// ---- DUTs/IO/Topology/RC40_A3_EK1122_E505EE87.TcDUT
{attribute 'GeneratedUsingTerminal: EK1122-0000-0018'}
{attribute addProperty BoxType "EK1122-0000-0018"}
{attribute addProperty Id "RC40_EPP_EPP1322_0001RC40_EPP_EPP1322_0001_ECA1E6F9120"}
{attribute addProperty CRC "3842371207"}
{attribute addProperty Size "120"}
{attribute addProperty Name "RC40_A3 (EK1122)"}
TYPE RC40_A3_EK1122_E505EE87 EXTENDS EK1122_1FC0878B :
STRUCT
    {attribute addProperty Name "RC40_EPP (EPP1322-0001)"}
    {attribute addProperty PreviousPort "RC40_A3 (EK1122) : D"}
    {attribute addProperty SyncUnit "default"}
    RC40_EPP_EPP1322_0001 : RC40_EPP_EPP1322_0001_ECA1E6F9;
END_STRUCT
END_TYPE

// ---- DUTs/IO/Topology/RC40_1_EK1100_B918F64D.TcDUT
{attribute 'GeneratedUsingTerminal: EK1100-0000-0018'}
{attribute addProperty BoxType "EK1100-0000-0018"}
{attribute addProperty Id "RC40_A2_EK1122RC40_A2_EK1122_EAFADCC873RC40_A3_EK1122RC40_A3_EK1122_E505EE87120RC40_A5_EL1809EL1809_32157CFD20RC40_A6_EL1809EL1809_32157CFD20RC40_A7_EL2809EL2809_2B6483BD19RC40_A8_EL2809EL2809_2B6483BD19RC40_A9_EL2809EL2809_2B6483BD19RC40_1_EndTerminal_EL9010EL9010_D29C20850"}
{attribute addProperty CRC "3105420877"}
{attribute addProperty Size "290"}
{attribute addProperty Name "RC40_1 (EK1100)"}
TYPE RC40_1_EK1100_B918F64D EXTENDS EK1100_1FC0878B :
STRUCT
    {attribute addProperty Name "RC40_A2 (EK1122)"}
    {attribute addProperty PreviousPort "RC40_1 (EK1100) : B"}
    {attribute addProperty SyncUnit "default"}
    RC40_A2_EK1122 : RC40_A2_EK1122_EAFADCC8;
    {attribute addProperty Name "RC40_A3 (EK1122)"}
    {attribute addProperty PreviousPort "RC40_A2 (EK1122) : C"}
    {attribute addProperty SyncUnit "default"}
    RC40_A3_EK1122 : RC40_A3_EK1122_E505EE87;
    {attribute addProperty Name "RC40_A5 (EL1809)"}
    {attribute addProperty PreviousPort "RC40_A3 (EK1122) : C"}
    {attribute addProperty SyncUnit "C40"}
    RC40_A5_EL1809 : EL1809_32157CFD;
    {attribute addProperty Name "RC40_A6 (EL1809)"}
    {attribute addProperty PreviousPort "RC40_A5 (EL1809) : B"}
    {attribute addProperty SyncUnit "C40"}
    RC40_A6_EL1809 : EL1809_32157CFD;
    {attribute addProperty Name "RC40_A7 (EL2809)"}
    {attribute addProperty PreviousPort "RC40_A6 (EL1809) : B"}
    {attribute addProperty SyncUnit "C40"}
    RC40_A7_EL2809 : EL2809_2B6483BD;
    {attribute addProperty Name "RC40_A8 (EL2809)"}
    {attribute addProperty PreviousPort "RC40_A7 (EL2809) : B"}
    {attribute addProperty SyncUnit "C40"}
    RC40_A8_EL2809 : EL2809_2B6483BD;
    {attribute addProperty Name "RC40_A9 (EL2809)"}
    {attribute addProperty PreviousPort "RC40_A8 (EL2809) : B"}
    {attribute addProperty SyncUnit "C40"}
    RC40_A9_EL2809 : EL2809_2B6483BD;
    {attribute addProperty Name "RC40_1_EndTerminal (EL9010)"}
    {attribute addProperty PreviousPort "RC40_A9 (EL2809) : B"}
    {attribute addProperty SyncUnit "default"}
    RC40_1_EndTerminal_EL9010 : EL9010_D29C2085;
END_STRUCT
END_TYPE

// ---- DUTs/IO/Topology/RC40_2_EK1100_ACF07759.TcDUT
{attribute 'GeneratedUsingTerminal: EK1100-0000-0018'}
{attribute addProperty BoxType "EK1100-0000-0018"}
{attribute addProperty Id "RC40_B1_EL7041_1000EL7041_86DE63E743RC40_B2_EL7041_1000EL7041_86DE63E743RC40_C11_EL7041_1000EL7041_86DE63E743RC40_C12_EL7041_1000EL7041_86DE63E743RC40_C21_EL7041_1000EL7041_86DE63E743RC40_C22_EL7041_1000EL7041_86DE63E743RC40_2_EndTerminal_EL9010EL9010_D29C20850"}
{attribute addProperty CRC "2901440345"}
{attribute addProperty Size "258"}
{attribute addProperty Name "RC40_2 (EK1100)"}
TYPE RC40_2_EK1100_ACF07759 EXTENDS EK1100_1FC0878B :
STRUCT
    {attribute addProperty Name "RC40_B1 (EL7041-1000)"}
    {attribute addProperty PreviousPort "RC40_2 (EK1100) : B"}
    {attribute addProperty SyncUnit "C40"}
    RC40_B1_EL7041_1000 : EL7041_86DE63E7;
    {attribute addProperty Name "RC40_B2 (EL7041-1000)"}
    {attribute addProperty PreviousPort "RC40_B1 (EL7041-1000) : B"}
    {attribute addProperty SyncUnit "C40"}
    RC40_B2_EL7041_1000 : EL7041_86DE63E7;
    {attribute addProperty Name "RC40_C11 (EL7041-1000)"}
    {attribute addProperty PreviousPort "RC40_B2 (EL7041-1000) : B"}
    {attribute addProperty SyncUnit "C40"}
    RC40_C11_EL7041_1000 : EL7041_86DE63E7;
    {attribute addProperty Name "RC40_C12 (EL7041-1000)"}
    {attribute addProperty PreviousPort "RC40_C11 (EL7041-1000) : B"}
    {attribute addProperty SyncUnit "C40"}
    RC40_C12_EL7041_1000 : EL7041_86DE63E7;
    {attribute addProperty Name "RC40_C21 (EL7041-1000)"}
    {attribute addProperty PreviousPort "RC40_C12 (EL7041-1000) : B"}
    {attribute addProperty SyncUnit "C40"}
    RC40_C21_EL7041_1000 : EL7041_86DE63E7;
    {attribute addProperty Name "RC40_C22 (EL7041-1000)"}
    {attribute addProperty PreviousPort "RC40_C21 (EL7041-1000) : B"}
    {attribute addProperty SyncUnit "C40"}
    RC40_C22_EL7041_1000 : EL7041_86DE63E7;
    {attribute addProperty Name "RC40_2_EndTerminal (EL9010)"}
    {attribute addProperty PreviousPort "RC40_C22 (EL7041-1000) : B"}
    {attribute addProperty SyncUnit "default"}
    RC40_2_EndTerminal_EL9010 : EL9010_D29C2085;
END_STRUCT
END_TYPE

// ---- DUTs/IO/Topology/R8_A9_EK1122_3EDD8752.TcDUT
{attribute 'GeneratedUsingTerminal: EK1122-0000-0018'}
{attribute addProperty BoxType "EK1122-0000-0018"}
{attribute addProperty Id "RC30_1_EK1100RC30_1_EK1100_B995809E290RC30_2_EK1100RC30_2_EK1100_8A0FE17C258RC40_1_EK1100RC40_1_EK1100_B918F64D290RC40_2_EK1100RC40_2_EK1100_ACF07759258"}
{attribute addProperty CRC "1054705490"}
{attribute addProperty Size "1096"}
{attribute addProperty Name "R8_A9 (EK1122)"}
TYPE R8_A9_EK1122_3EDD8752 EXTENDS EK1122_1FC0878B :
STRUCT
    {attribute addProperty Name "RC30_1 (EK1100)"}
    {attribute addProperty PreviousPort "R8_A9 (EK1122) : D"}
    {attribute addProperty SyncUnit "default"}
    RC30_1_EK1100 : RC30_1_EK1100_B995809E;
    {attribute addProperty Name "RC30_2 (EK1100)"}
    {attribute addProperty PreviousPort "RC30_1 (EK1100) : C"}
    {attribute addProperty SyncUnit "default"}
    RC30_2_EK1100 : RC30_2_EK1100_8A0FE17C;
    {attribute addProperty Name "RC40_1 (EK1100)"}
    {attribute addProperty PreviousPort "R8_A9 (EK1122) : B"}
    {attribute addProperty SyncUnit "default"}
    RC40_1_EK1100 : RC40_1_EK1100_B918F64D;
    {attribute addProperty Name "RC40_2 (EK1100)"}
    {attribute addProperty PreviousPort "RC40_1 (EK1100) : C"}
    {attribute addProperty SyncUnit "default"}
    RC40_2_EK1100 : RC40_2_EK1100_ACF07759;
END_STRUCT
END_TYPE

// ---- DUTs/IO/Topology/RC50_A2_EK1122_AE8686CC.TcDUT
{attribute 'GeneratedUsingTerminal: EK1122-0000-0018'}
{attribute addProperty BoxType "EK1122-0000-0018"}
{attribute addProperty Id "RC50_VI_AES_D_BC_ECAT_xAES_A3B0707168RC50_SAFETY_Flexi_Soft_EtherCAT_GatewayFlexi_Soft_EtherCAT_Gateway_DE394EDD5"}
{attribute addProperty CRC "2928051916"}
{attribute addProperty Size "73"}
{attribute addProperty Name "RC50_A2 (EK1122)"}
TYPE RC50_A2_EK1122_AE8686CC EXTENDS EK1122_1FC0878B :
STRUCT
    {attribute addProperty Name "RC50_VI (AES-D-BC-ECAT)"}
    {attribute addProperty PreviousPort "RC50_A2 (EK1122) : D"}
    {attribute addProperty SyncUnit "C50"}
    RC50_VI_AES_D_BC_ECAT_x : AES_A3B07071;
    {attribute addProperty Name "RC50_SAFETY (Flexi Soft EtherCAT Gateway)"}
    {attribute addProperty PreviousPort "RC50_A2 (EK1122) : B"}
    {attribute addProperty SyncUnit "C50"}
    RC50_SAFETY_Flexi_Soft_EtherCAT_Gateway : Flexi_Soft_EtherCAT_Gateway_DE394EDD;
END_STRUCT
END_TYPE

// ---- DUTs/IO/Topology/RC50_EPP_EPP1322_0001_58A8DEC2.TcDUT
{attribute 'GeneratedUsingTerminal: EPP1322-0001-0017'}
{attribute addProperty BoxType "EPP1322-0001-0017"}
{attribute addProperty Id "RC50_AB1_EPP1008_0001EPP1008_78E8D3DD12RC50_AB2_EPP1008_0001EPP1008_78E8D3DD12RC50_AB6_EPP1008_0001EPP1008_78E8D3DD12RC50_AB3_EPP1008_0001EPP1008_78E8D3DD12RC50_AB4_EPP1008_0001EPP1008_78E8D3DD12RC50_AB7_EPP1008_0001EPP1008_78E8D3DD12RC50_AB9_EPP1008_0001EPP1008_78E8D3DD12RC50_AB10_EPP1008_0001EPP1008_78E8D3DD12RC50_AB8_EPP1008_0001EPP1008_78E8D3DD12RC50_AB5_EPP1008_0001EPP1008_78E8D3DD12"}
{attribute addProperty CRC "1487462082"}
{attribute addProperty Size "120"}
{attribute addProperty Name "RC50_EPP (EPP1322-0001)"}
TYPE RC50_EPP_EPP1322_0001_58A8DEC2 EXTENDS EPP1322_1FC0878B :
STRUCT
    {attribute addProperty Name "RC50_AB1 (EPP1008-0001)"}
    {attribute addProperty PreviousPort "RC50_EPP (EPP1322-0001) : D"}
    {attribute addProperty SyncUnit "C50"}
    RC50_AB1_EPP1008_0001 : EPP1008_78E8D3DD;
    {attribute addProperty Name "RC50_AB2 (EPP1008-0001)"}
    {attribute addProperty PreviousPort "RC50_AB1 (EPP1008-0001) : B"}
    {attribute addProperty SyncUnit "C50"}
    RC50_AB2_EPP1008_0001 : EPP1008_78E8D3DD;
    {attribute addProperty Name "RC50_AB6 (EPP1008-0001)"}
    {attribute addProperty PreviousPort "RC50_AB2 (EPP1008-0001) : B"}
    {attribute addProperty SyncUnit "C50"}
    RC50_AB6_EPP1008_0001 : EPP1008_78E8D3DD;
    {attribute addProperty Name "RC50_AB3 (EPP1008-0001)"}
    {attribute addProperty PreviousPort "RC50_AB6 (EPP1008-0001) : B"}
    {attribute addProperty SyncUnit "C50"}
    RC50_AB3_EPP1008_0001 : EPP1008_78E8D3DD;
    {attribute addProperty Name "RC50_AB4 (EPP1008-0001)"}
    {attribute addProperty PreviousPort "RC50_AB3 (EPP1008-0001) : B"}
    {attribute addProperty SyncUnit "C50"}
    RC50_AB4_EPP1008_0001 : EPP1008_78E8D3DD;
    {attribute addProperty Name "RC50_AB7 (EPP1008-0001)"}
    {attribute addProperty PreviousPort "RC50_EPP (EPP1322-0001) : B"}
    {attribute addProperty SyncUnit "C50"}
    RC50_AB7_EPP1008_0001 : EPP1008_78E8D3DD;
    {attribute addProperty Name "RC50_AB9 (EPP1008-0001)"}
    {attribute addProperty PreviousPort "RC50_AB7 (EPP1008-0001) : B"}
    {attribute addProperty SyncUnit "C50"}
    RC50_AB9_EPP1008_0001 : EPP1008_78E8D3DD;
    {attribute addProperty Name "RC50_AB10 (EPP1008-0001)"}
    {attribute addProperty PreviousPort "RC50_AB9 (EPP1008-0001) : B"}
    {attribute addProperty SyncUnit "C50"}
    RC50_AB10_EPP1008_0001 : EPP1008_78E8D3DD;
    {attribute addProperty Name "RC50_AB8 (EPP1008-0001)"}
    {attribute addProperty PreviousPort "RC50_AB10 (EPP1008-0001) : B"}
    {attribute addProperty SyncUnit "C50"}
    RC50_AB8_EPP1008_0001 : EPP1008_78E8D3DD;
    {attribute addProperty Name "RC50_AB5 (EPP1008-0001)"}
    {attribute addProperty PreviousPort "RC50_AB8 (EPP1008-0001) : B"}
    {attribute addProperty SyncUnit "C50"}
    RC50_AB5_EPP1008_0001 : EPP1008_78E8D3DD;
END_STRUCT
END_TYPE

// ---- DUTs/IO/Topology/RC50_A3_EK1122_7F1D927D.TcDUT
{attribute 'GeneratedUsingTerminal: EK1122-0000-0018'}
{attribute addProperty BoxType "EK1122-0000-0018"}
{attribute addProperty Id "RC50_EPP_EPP1322_0001RC50_EPP_EPP1322_0001_58A8DEC2120"}
{attribute addProperty CRC "2132644477"}
{attribute addProperty Size "120"}
{attribute addProperty Name "RC50_A3 (EK1122)"}
TYPE RC50_A3_EK1122_7F1D927D EXTENDS EK1122_1FC0878B :
STRUCT
    {attribute addProperty Name "RC50_EPP (EPP1322-0001)"}
    {attribute addProperty PreviousPort "RC50_A3 (EK1122) : D"}
    {attribute addProperty SyncUnit "default"}
    RC50_EPP_EPP1322_0001 : RC50_EPP_EPP1322_0001_58A8DEC2;
END_STRUCT
END_TYPE

// ---- DUTs/IO/Topology/RC50_1_EK1100_D6E64946.TcDUT
{attribute 'GeneratedUsingTerminal: EK1100-0000-0018'}
{attribute addProperty BoxType "EK1100-0000-0018"}
{attribute addProperty Id "RC50_A2_EK1122RC50_A2_EK1122_AE8686CC73RC50_A3_EK1122RC50_A3_EK1122_7F1D927D120RC50_A5_EL1809EL1809_32157CFD20RC50_A6_EL1809EL1809_32157CFD20RC50_A7_EL2809EL2809_2B6483BD19RC50_A8_EL2809EL2809_2B6483BD19RC50_A9_EL2809EL2809_2B6483BD19RC50_1_EndTerminal_EL9010EL9010_D29C20850"}
{attribute addProperty CRC "3605416262"}
{attribute addProperty Size "290"}
{attribute addProperty Name "RC50_1 (EK1100)"}
TYPE RC50_1_EK1100_D6E64946 EXTENDS EK1100_1FC0878B :
STRUCT
    {attribute addProperty Name "RC50_A2 (EK1122)"}
    {attribute addProperty PreviousPort "RC50_1 (EK1100) : B"}
    {attribute addProperty SyncUnit "default"}
    RC50_A2_EK1122 : RC50_A2_EK1122_AE8686CC;
    {attribute addProperty Name "RC50_A3 (EK1122)"}
    {attribute addProperty PreviousPort "RC50_A2 (EK1122) : C"}
    {attribute addProperty SyncUnit "default"}
    RC50_A3_EK1122 : RC50_A3_EK1122_7F1D927D;
    {attribute addProperty Name "RC50_A5 (EL1809)"}
    {attribute addProperty PreviousPort "RC50_A3 (EK1122) : C"}
    {attribute addProperty SyncUnit "C50"}
    RC50_A5_EL1809 : EL1809_32157CFD;
    {attribute addProperty Name "RC50_A6 (EL1809)"}
    {attribute addProperty PreviousPort "RC50_A5 (EL1809) : B"}
    {attribute addProperty SyncUnit "C50"}
    RC50_A6_EL1809 : EL1809_32157CFD;
    {attribute addProperty Name "RC50_A7 (EL2809)"}
    {attribute addProperty PreviousPort "RC50_A6 (EL1809) : B"}
    {attribute addProperty SyncUnit "C50"}
    RC50_A7_EL2809 : EL2809_2B6483BD;
    {attribute addProperty Name "RC50_A8 (EL2809)"}
    {attribute addProperty PreviousPort "RC50_A7 (EL2809) : B"}
    {attribute addProperty SyncUnit "C50"}
    RC50_A8_EL2809 : EL2809_2B6483BD;
    {attribute addProperty Name "RC50_A9 (EL2809)"}
    {attribute addProperty PreviousPort "RC50_A8 (EL2809) : B"}
    {attribute addProperty SyncUnit "C50"}
    RC50_A9_EL2809 : EL2809_2B6483BD;
    {attribute addProperty Name "RC50_1_EndTerminal (EL9010)"}
    {attribute addProperty PreviousPort "RC50_A9 (EL2809) : B"}
    {attribute addProperty SyncUnit "default"}
    RC50_1_EndTerminal_EL9010 : EL9010_D29C2085;
END_STRUCT
END_TYPE

// ---- DUTs/IO/Topology/RC50_2_EK1100_7854232C.TcDUT
{attribute 'GeneratedUsingTerminal: EK1100-0000-0018'}
{attribute addProperty BoxType "EK1100-0000-0018"}
{attribute addProperty Id "RC50_B1_EL7041_1000EL7041_86DE63E743RC50_B2_EL7041_1000EL7041_86DE63E743RC50_C11_EL7041_1000EL7041_86DE63E743RC50_C12_EL7041_1000EL7041_86DE63E743RC50_C21_EL7041_1000EL7041_86DE63E743RC50_C22_EL7041_1000EL7041_86DE63E743RC50_2_EndTerminal_EL9010EL9010_D29C20850"}
{attribute addProperty CRC "2018779948"}
{attribute addProperty Size "258"}
{attribute addProperty Name "RC50_2 (EK1100)"}
TYPE RC50_2_EK1100_7854232C EXTENDS EK1100_1FC0878B :
STRUCT
    {attribute addProperty Name "RC50_B1 (EL7041-1000)"}
    {attribute addProperty PreviousPort "RC50_2 (EK1100) : B"}
    {attribute addProperty SyncUnit "C50"}
    RC50_B1_EL7041_1000 : EL7041_86DE63E7;
    {attribute addProperty Name "RC50_B2 (EL7041-1000)"}
    {attribute addProperty PreviousPort "RC50_B1 (EL7041-1000) : B"}
    {attribute addProperty SyncUnit "C50"}
    RC50_B2_EL7041_1000 : EL7041_86DE63E7;
    {attribute addProperty Name "RC50_C11 (EL7041-1000)"}
    {attribute addProperty PreviousPort "RC50_B2 (EL7041-1000) : B"}
    {attribute addProperty SyncUnit "C50"}
    RC50_C11_EL7041_1000 : EL7041_86DE63E7;
    {attribute addProperty Name "RC50_C12 (EL7041-1000)"}
    {attribute addProperty PreviousPort "RC50_C11 (EL7041-1000) : B"}
    {attribute addProperty SyncUnit "C50"}
    RC50_C12_EL7041_1000 : EL7041_86DE63E7;
    {attribute addProperty Name "RC50_C21 (EL7041-1000)"}
    {attribute addProperty PreviousPort "RC50_C12 (EL7041-1000) : B"}
    {attribute addProperty SyncUnit "C50"}
    RC50_C21_EL7041_1000 : EL7041_86DE63E7;
    {attribute addProperty Name "RC50_C22 (EL7041-1000)"}
    {attribute addProperty PreviousPort "RC50_C21 (EL7041-1000) : B"}
    {attribute addProperty SyncUnit "C50"}
    RC50_C22_EL7041_1000 : EL7041_86DE63E7;
    {attribute addProperty Name "RC50_2_EndTerminal (EL9010)"}
    {attribute addProperty PreviousPort "RC50_C22 (EL7041-1000) : B"}
    {attribute addProperty SyncUnit "default"}
    RC50_2_EndTerminal_EL9010 : EL9010_D29C2085;
END_STRUCT
END_TYPE

// ---- DUTs/IO/Topology/RC60_A2_EK1122_620268C0.TcDUT
{attribute 'GeneratedUsingTerminal: EK1122-0000-0018'}
{attribute addProperty BoxType "EK1122-0000-0018"}
{attribute addProperty Id "RC60_VI_AES_D_BC_ECAT_xAES_A3B0707168RC60_SAFETY_Flexi_Soft_EtherCAT_GatewayFlexi_Soft_EtherCAT_Gateway_DE394EDD5"}
{attribute addProperty CRC "1644325056"}
{attribute addProperty Size "73"}
{attribute addProperty Name "RC60_A2 (EK1122)"}
TYPE RC60_A2_EK1122_620268C0 EXTENDS EK1122_1FC0878B :
STRUCT
    {attribute addProperty Name "RC60_VI (AES-D-BC-ECAT)"}
    {attribute addProperty PreviousPort "RC60_A2 (EK1122) : D"}
    {attribute addProperty SyncUnit "C60"}
    RC60_VI_AES_D_BC_ECAT_x : AES_A3B07071;
    {attribute addProperty Name "RC60_SAFETY (Flexi Soft EtherCAT Gateway)"}
    {attribute addProperty PreviousPort "RC60_A2 (EK1122) : B"}
    {attribute addProperty SyncUnit "C60"}
    RC60_SAFETY_Flexi_Soft_EtherCAT_Gateway : Flexi_Soft_EtherCAT_Gateway_DE394EDD;
END_STRUCT
END_TYPE

// ---- DUTs/IO/Topology/RC60_EPP_EPP1322_0001_80728B38.TcDUT
{attribute 'GeneratedUsingTerminal: EPP1322-0001-0017'}
{attribute addProperty BoxType "EPP1322-0001-0017"}
{attribute addProperty Id "RC60_AB1_EPP1008_0001EPP1008_78E8D3DD12RC60_AB2_EPP1008_0001EPP1008_78E8D3DD12RC60_AB6_EPP1008_0001EPP1008_78E8D3DD12RC60_AB3_EPP1008_0001EPP1008_78E8D3DD12RC60_AB4_EPP1008_0001EPP1008_78E8D3DD12RC60_AB7_EPP1008_0001EPP1008_78E8D3DD12RC60_AB9_EPP1008_0001EPP1008_78E8D3DD12RC60_AB10_EPP1008_0001EPP1008_78E8D3DD12RC60_AB8_EPP1008_0001EPP1008_78E8D3DD12RC60_AB5_EPP1008_0001EPP1008_78E8D3DD12"}
{attribute addProperty CRC "2154990392"}
{attribute addProperty Size "120"}
{attribute addProperty Name "RC60_EPP (EPP1322-0001)"}
TYPE RC60_EPP_EPP1322_0001_80728B38 EXTENDS EPP1322_1FC0878B :
STRUCT
    {attribute addProperty Name "RC60_AB1 (EPP1008-0001)"}
    {attribute addProperty PreviousPort "RC60_EPP (EPP1322-0001) : D"}
    {attribute addProperty SyncUnit "C60"}
    RC60_AB1_EPP1008_0001 : EPP1008_78E8D3DD;
    {attribute addProperty Name "RC60_AB2 (EPP1008-0001)"}
    {attribute addProperty PreviousPort "RC60_AB1 (EPP1008-0001) : B"}
    {attribute addProperty SyncUnit "C60"}
    RC60_AB2_EPP1008_0001 : EPP1008_78E8D3DD;
    {attribute addProperty Name "RC60_AB6 (EPP1008-0001)"}
    {attribute addProperty PreviousPort "RC60_AB2 (EPP1008-0001) : B"}
    {attribute addProperty SyncUnit "C60"}
    RC60_AB6_EPP1008_0001 : EPP1008_78E8D3DD;
    {attribute addProperty Name "RC60_AB3 (EPP1008-0001)"}
    {attribute addProperty PreviousPort "RC60_AB6 (EPP1008-0001) : B"}
    {attribute addProperty SyncUnit "C60"}
    RC60_AB3_EPP1008_0001 : EPP1008_78E8D3DD;
    {attribute addProperty Name "RC60_AB4 (EPP1008-0001)"}
    {attribute addProperty PreviousPort "RC60_AB3 (EPP1008-0001) : B"}
    {attribute addProperty SyncUnit "C60"}
    RC60_AB4_EPP1008_0001 : EPP1008_78E8D3DD;
    {attribute addProperty Name "RC60_AB7 (EPP1008-0001)"}
    {attribute addProperty PreviousPort "RC60_EPP (EPP1322-0001) : B"}
    {attribute addProperty SyncUnit "C60"}
    RC60_AB7_EPP1008_0001 : EPP1008_78E8D3DD;
    {attribute addProperty Name "RC60_AB9 (EPP1008-0001)"}
    {attribute addProperty PreviousPort "RC60_AB7 (EPP1008-0001) : B"}
    {attribute addProperty SyncUnit "C60"}
    RC60_AB9_EPP1008_0001 : EPP1008_78E8D3DD;
    {attribute addProperty Name "RC60_AB10 (EPP1008-0001)"}
    {attribute addProperty PreviousPort "RC60_AB9 (EPP1008-0001) : B"}
    {attribute addProperty SyncUnit "C60"}
    RC60_AB10_EPP1008_0001 : EPP1008_78E8D3DD;
    {attribute addProperty Name "RC60_AB8 (EPP1008-0001)"}
    {attribute addProperty PreviousPort "RC60_AB10 (EPP1008-0001) : B"}
    {attribute addProperty SyncUnit "C60"}
    RC60_AB8_EPP1008_0001 : EPP1008_78E8D3DD;
    {attribute addProperty Name "RC60_AB5 (EPP1008-0001)"}
    {attribute addProperty PreviousPort "RC60_AB8 (EPP1008-0001) : B"}
    {attribute addProperty SyncUnit "C60"}
    RC60_AB5_EPP1008_0001 : EPP1008_78E8D3DD;
END_STRUCT
END_TYPE

// ---- DUTs/IO/Topology/RC60_A3_EK1122_0BEA55B5.TcDUT
{attribute 'GeneratedUsingTerminal: EK1122-0000-0018'}
{attribute addProperty BoxType "EK1122-0000-0018"}
{attribute addProperty Id "RC60_EPP_EPP1322_0001RC60_EPP_EPP1322_0001_80728B38120"}
{attribute addProperty CRC "199906741"}
{attribute addProperty Size "120"}
{attribute addProperty Name "RC60_A3 (EK1122)"}
TYPE RC60_A3_EK1122_0BEA55B5 EXTENDS EK1122_1FC0878B :
STRUCT
    {attribute addProperty Name "RC60_EPP (EPP1322-0001)"}
    {attribute addProperty PreviousPort "RC60_A3 (EK1122) : D"}
    {attribute addProperty SyncUnit "default"}
    RC60_EPP_EPP1322_0001 : RC60_EPP_EPP1322_0001_80728B38;
END_STRUCT
END_TYPE

// ---- DUTs/IO/Topology/RC60_1_EK1100_9BABA6E0.TcDUT
{attribute 'GeneratedUsingTerminal: EK1100-0000-0018'}
{attribute addProperty BoxType "EK1100-0000-0018"}
{attribute addProperty Id "RC60_A2_EK1122RC60_A2_EK1122_620268C073RC60_A3_EK1122RC60_A3_EK1122_0BEA55B5120RC60_A5_EL1809EL1809_32157CFD20RC60_A6_EL1809EL1809_32157CFD20RC60_A7_EL2809EL2809_2B6483BD19RC60_A8_EL2809EL2809_2B6483BD19RC60_A9_EL2809EL2809_2B6483BD19RC60_1_EndTerminal_EL9010EL9010_D29C20850"}
{attribute addProperty CRC "2611717856"}
{attribute addProperty Size "290"}
{attribute addProperty Name "RC60_1 (EK1100)"}
TYPE RC60_1_EK1100_9BABA6E0 EXTENDS EK1100_1FC0878B :
STRUCT
    {attribute addProperty Name "RC60_A2 (EK1122)"}
    {attribute addProperty PreviousPort "RC60_1 (EK1100) : B"}
    {attribute addProperty SyncUnit "default"}
    RC60_A2_EK1122 : RC60_A2_EK1122_620268C0;
    {attribute addProperty Name "RC60_A3 (EK1122)"}
    {attribute addProperty PreviousPort "RC60_A2 (EK1122) : C"}
    {attribute addProperty SyncUnit "default"}
    RC60_A3_EK1122 : RC60_A3_EK1122_0BEA55B5;
    {attribute addProperty Name "RC60_A5 (EL1809)"}
    {attribute addProperty PreviousPort "RC60_A3 (EK1122) : C"}
    {attribute addProperty SyncUnit "C60"}
    RC60_A5_EL1809 : EL1809_32157CFD;
    {attribute addProperty Name "RC60_A6 (EL1809)"}
    {attribute addProperty PreviousPort "RC60_A5 (EL1809) : B"}
    {attribute addProperty SyncUnit "C60"}
    RC60_A6_EL1809 : EL1809_32157CFD;
    {attribute addProperty Name "RC60_A7 (EL2809)"}
    {attribute addProperty PreviousPort "RC60_A6 (EL1809) : B"}
    {attribute addProperty SyncUnit "C60"}
    RC60_A7_EL2809 : EL2809_2B6483BD;
    {attribute addProperty Name "RC60_A8 (EL2809)"}
    {attribute addProperty PreviousPort "RC60_A7 (EL2809) : B"}
    {attribute addProperty SyncUnit "C60"}
    RC60_A8_EL2809 : EL2809_2B6483BD;
    {attribute addProperty Name "RC60_A9 (EL2809)"}
    {attribute addProperty PreviousPort "RC60_A8 (EL2809) : B"}
    {attribute addProperty SyncUnit "C60"}
    RC60_A9_EL2809 : EL2809_2B6483BD;
    {attribute addProperty Name "RC60_1_EndTerminal (EL9010)"}
    {attribute addProperty PreviousPort "RC60_A9 (EL2809) : B"}
    {attribute addProperty SyncUnit "default"}
    RC60_1_EndTerminal_EL9010 : EL9010_D29C2085;
END_STRUCT
END_TYPE

// ---- DUTs/IO/Topology/RC60_2_EK1100_0179C204.TcDUT
{attribute 'GeneratedUsingTerminal: EK1100-0000-0018'}
{attribute addProperty BoxType "EK1100-0000-0018"}
{attribute addProperty Id "RC60_B1_EL7041_1000EL7041_86DE63E743RC60_B2_EL7041_1000EL7041_86DE63E743RC60_C11_EL7041_1000EL7041_86DE63E743RC60_C12_EL7041_1000EL7041_86DE63E743RC60_C21_EL7041_1000EL7041_86DE63E743RC60_C22_EL7041_1000EL7041_86DE63E743RC60_2_EndTerminal_EL9010EL9010_D29C20850"}
{attribute addProperty CRC "24756740"}
{attribute addProperty Size "258"}
{attribute addProperty Name "RC60_2 (EK1100)"}
TYPE RC60_2_EK1100_0179C204 EXTENDS EK1100_1FC0878B :
STRUCT
    {attribute addProperty Name "RC60_B1 (EL7041-1000)"}
    {attribute addProperty PreviousPort "RC60_2 (EK1100) : B"}
    {attribute addProperty SyncUnit "C60"}
    RC60_B1_EL7041_1000 : EL7041_86DE63E7;
    {attribute addProperty Name "RC60_B2 (EL7041-1000)"}
    {attribute addProperty PreviousPort "RC60_B1 (EL7041-1000) : B"}
    {attribute addProperty SyncUnit "C60"}
    RC60_B2_EL7041_1000 : EL7041_86DE63E7;
    {attribute addProperty Name "RC60_C11 (EL7041-1000)"}
    {attribute addProperty PreviousPort "RC60_B2 (EL7041-1000) : B"}
    {attribute addProperty SyncUnit "C60"}
    RC60_C11_EL7041_1000 : EL7041_86DE63E7;
    {attribute addProperty Name "RC60_C12 (EL7041-1000)"}
    {attribute addProperty PreviousPort "RC60_C11 (EL7041-1000) : B"}
    {attribute addProperty SyncUnit "C60"}
    RC60_C12_EL7041_1000 : EL7041_86DE63E7;
    {attribute addProperty Name "RC60_C21 (EL7041-1000)"}
    {attribute addProperty PreviousPort "RC60_C12 (EL7041-1000) : B"}
    {attribute addProperty SyncUnit "C60"}
    RC60_C21_EL7041_1000 : EL7041_86DE63E7;
    {attribute addProperty Name "RC60_C22 (EL7041-1000)"}
    {attribute addProperty PreviousPort "RC60_C21 (EL7041-1000) : B"}
    {attribute addProperty SyncUnit "C60"}
    RC60_C22_EL7041_1000 : EL7041_86DE63E7;
    {attribute addProperty Name "RC60_2_EndTerminal (EL9010)"}
    {attribute addProperty PreviousPort "RC60_C22 (EL7041-1000) : B"}
    {attribute addProperty SyncUnit "default"}
    RC60_2_EndTerminal_EL9010 : EL9010_D29C2085;
END_STRUCT
END_TYPE

// ---- DUTs/IO/Topology/R8_A10_EK1122_484442E0.TcDUT
{attribute 'GeneratedUsingTerminal: EK1122-0000-0018'}
{attribute addProperty BoxType "EK1122-0000-0018"}
{attribute addProperty Id "RC50_1_EK1100RC50_1_EK1100_D6E64946290RC50_2_EK1100RC50_2_EK1100_7854232C258RC60_1_EK1100RC60_1_EK1100_9BABA6E0290RC60_2_EK1100RC60_2_EK1100_0179C204258"}
{attribute addProperty CRC "1212433120"}
{attribute addProperty Size "1096"}
{attribute addProperty Name "R8_A10 (EK1122)"}
TYPE R8_A10_EK1122_484442E0 EXTENDS EK1122_1FC0878B :
STRUCT
    {attribute addProperty Name "RC50_1 (EK1100)"}
    {attribute addProperty PreviousPort "R8_A10 (EK1122) : D"}
    {attribute addProperty SyncUnit "default"}
    RC50_1_EK1100 : RC50_1_EK1100_D6E64946;
    {attribute addProperty Name "RC50_2 (EK1100)"}
    {attribute addProperty PreviousPort "RC50_1 (EK1100) : C"}
    {attribute addProperty SyncUnit "default"}
    RC50_2_EK1100 : RC50_2_EK1100_7854232C;
    {attribute addProperty Name "RC60_1 (EK1100)"}
    {attribute addProperty PreviousPort "R8_A10 (EK1122) : B"}
    {attribute addProperty SyncUnit "default"}
    RC60_1_EK1100 : RC60_1_EK1100_9BABA6E0;
    {attribute addProperty Name "RC60_2 (EK1100)"}
    {attribute addProperty PreviousPort "RC60_1 (EK1100) : C"}
    {attribute addProperty SyncUnit "default"}
    RC60_2_EK1100 : RC60_2_EK1100_0179C204;
END_STRUCT
END_TYPE

// ---- DUTs/IO/Topology/RC70_A2_EK1122_267E32C4.TcDUT
{attribute 'GeneratedUsingTerminal: EK1122-0000-0018'}
{attribute addProperty BoxType "EK1122-0000-0018"}
{attribute addProperty Id "RC70_VI_AES_D_BC_ECAT_xAES_A3B0707168RC70_SAFETY_Flexi_Soft_EtherCAT_GatewayFlexi_Soft_EtherCAT_Gateway_DE394EDD5"}
{attribute addProperty CRC "645804740"}
{attribute addProperty Size "73"}
{attribute addProperty Name "RC70_A2 (EK1122)"}
TYPE RC70_A2_EK1122_267E32C4 EXTENDS EK1122_1FC0878B :
STRUCT
    {attribute addProperty Name "RC70_VI (AES-D-BC-ECAT)"}
    {attribute addProperty PreviousPort "RC70_A2 (EK1122) : D"}
    {attribute addProperty SyncUnit "C70"}
    RC70_VI_AES_D_BC_ECAT_x : AES_A3B07071;
    {attribute addProperty Name "RC70_SAFETY (Flexi Soft EtherCAT Gateway)"}
    {attribute addProperty PreviousPort "RC70_A2 (EK1122) : B"}
    {attribute addProperty SyncUnit "C70"}
    RC70_SAFETY_Flexi_Soft_EtherCAT_Gateway : Flexi_Soft_EtherCAT_Gateway_DE394EDD;
END_STRUCT
END_TYPE

// ---- DUTs/IO/Topology/RC70_EPP_EPP1322_0001_347BB303.TcDUT
{attribute 'GeneratedUsingTerminal: EPP1322-0001-0017'}
{attribute addProperty BoxType "EPP1322-0001-0017"}
{attribute addProperty Id "RC70_AB1_EPP1008_0001EPP1008_78E8D3DD12RC70_AB2_EPP1008_0001EPP1008_78E8D3DD12RC70_AB6_EPP1008_0001EPP1008_78E8D3DD12RC70_AB3_EPP1008_0001EPP1008_78E8D3DD12RC70_AB4_EPP1008_0001EPP1008_78E8D3DD12RC70_AB7_EPP1008_0001EPP1008_78E8D3DD12RC70_AB9_EPP1008_0001EPP1008_78E8D3DD12RC70_AB10_EPP1008_0001EPP1008_78E8D3DD12RC70_AB8_EPP1008_0001EPP1008_78E8D3DD12RC70_AB5_EPP1008_0001EPP1008_78E8D3DD12"}
{attribute addProperty CRC "880521987"}
{attribute addProperty Size "120"}
{attribute addProperty Name "RC70_EPP (EPP1322-0001)"}
TYPE RC70_EPP_EPP1322_0001_347BB303 EXTENDS EPP1322_1FC0878B :
STRUCT
    {attribute addProperty Name "RC70_AB1 (EPP1008-0001)"}
    {attribute addProperty PreviousPort "RC70_EPP (EPP1322-0001) : D"}
    {attribute addProperty SyncUnit "C70"}
    RC70_AB1_EPP1008_0001 : EPP1008_78E8D3DD;
    {attribute addProperty Name "RC70_AB2 (EPP1008-0001)"}
    {attribute addProperty PreviousPort "RC70_AB1 (EPP1008-0001) : B"}
    {attribute addProperty SyncUnit "C70"}
    RC70_AB2_EPP1008_0001 : EPP1008_78E8D3DD;
    {attribute addProperty Name "RC70_AB6 (EPP1008-0001)"}
    {attribute addProperty PreviousPort "RC70_AB2 (EPP1008-0001) : B"}
    {attribute addProperty SyncUnit "C70"}
    RC70_AB6_EPP1008_0001 : EPP1008_78E8D3DD;
    {attribute addProperty Name "RC70_AB3 (EPP1008-0001)"}
    {attribute addProperty PreviousPort "RC70_AB6 (EPP1008-0001) : B"}
    {attribute addProperty SyncUnit "C70"}
    RC70_AB3_EPP1008_0001 : EPP1008_78E8D3DD;
    {attribute addProperty Name "RC70_AB4 (EPP1008-0001)"}
    {attribute addProperty PreviousPort "RC70_AB3 (EPP1008-0001) : B"}
    {attribute addProperty SyncUnit "C70"}
    RC70_AB4_EPP1008_0001 : EPP1008_78E8D3DD;
    {attribute addProperty Name "RC70_AB7 (EPP1008-0001)"}
    {attribute addProperty PreviousPort "RC70_EPP (EPP1322-0001) : B"}
    {attribute addProperty SyncUnit "C70"}
    RC70_AB7_EPP1008_0001 : EPP1008_78E8D3DD;
    {attribute addProperty Name "RC70_AB9 (EPP1008-0001)"}
    {attribute addProperty PreviousPort "RC70_AB7 (EPP1008-0001) : B"}
    {attribute addProperty SyncUnit "C70"}
    RC70_AB9_EPP1008_0001 : EPP1008_78E8D3DD;
    {attribute addProperty Name "RC70_AB10 (EPP1008-0001)"}
    {attribute addProperty PreviousPort "RC70_AB9 (EPP1008-0001) : B"}
    {attribute addProperty SyncUnit "C70"}
    RC70_AB10_EPP1008_0001 : EPP1008_78E8D3DD;
    {attribute addProperty Name "RC70_AB8 (EPP1008-0001)"}
    {attribute addProperty PreviousPort "RC70_AB10 (EPP1008-0001) : B"}
    {attribute addProperty SyncUnit "C70"}
    RC70_AB8_EPP1008_0001 : EPP1008_78E8D3DD;
    {attribute addProperty Name "RC70_AB5 (EPP1008-0001)"}
    {attribute addProperty PreviousPort "RC70_AB8 (EPP1008-0001) : B"}
    {attribute addProperty SyncUnit "C70"}
    RC70_AB5_EPP1008_0001 : EPP1008_78E8D3DD;
END_STRUCT
END_TYPE

// ---- DUTs/IO/Topology/RC70_A3_EK1122_27C9256F.TcDUT
{attribute 'GeneratedUsingTerminal: EK1122-0000-0018'}
{attribute addProperty BoxType "EK1122-0000-0018"}
{attribute addProperty Id "RC70_EPP_EPP1322_0001RC70_EPP_EPP1322_0001_347BB303120"}
{attribute addProperty CRC "667493743"}
{attribute addProperty Size "120"}
{attribute addProperty Name "RC70_A3 (EK1122)"}
TYPE RC70_A3_EK1122_27C9256F EXTENDS EK1122_1FC0878B :
STRUCT
    {attribute addProperty Name "RC70_EPP (EPP1322-0001)"}
    {attribute addProperty PreviousPort "RC70_A3 (EK1122) : D"}
    {attribute addProperty SyncUnit "default"}
    RC70_EPP_EPP1322_0001 : RC70_EPP_EPP1322_0001_347BB303;
END_STRUCT
END_TYPE

// ---- DUTs/IO/Topology/RC70_1_EK1100_B905944A.TcDUT
{attribute 'GeneratedUsingTerminal: EK1100-0000-0018'}
{attribute addProperty BoxType "EK1100-0000-0018"}
{attribute addProperty Id "RC70_A2_EK1122RC70_A2_EK1122_267E32C473RC70_A3_EK1122RC70_A3_EK1122_27C9256F120RC70_A5_EL1809EL1809_32157CFD20RC70_A6_EL1809EL1809_32157CFD20RC70_A7_EL2809EL2809_2B6483BD19RC70_A8_EL2809EL2809_2B6483BD19RC70_A9_EL2809EL2809_2B6483BD19RC70_1_EndTerminal_EL9010EL9010_D29C20850"}
{attribute addProperty CRC "3104150602"}
{attribute addProperty Size "290"}
{attribute addProperty Name "RC70_1 (EK1100)"}
TYPE RC70_1_EK1100_B905944A EXTENDS EK1100_1FC0878B :
STRUCT
    {attribute addProperty Name "RC70_A2 (EK1122)"}
    {attribute addProperty PreviousPort "RC70_1 (EK1100) : B"}
    {attribute addProperty SyncUnit "default"}
    RC70_A2_EK1122 : RC70_A2_EK1122_267E32C4;
    {attribute addProperty Name "RC70_A3 (EK1122)"}
    {attribute addProperty PreviousPort "RC70_A2 (EK1122) : C"}
    {attribute addProperty SyncUnit "default"}
    RC70_A3_EK1122 : RC70_A3_EK1122_27C9256F;
    {attribute addProperty Name "RC70_A5 (EL1809)"}
    {attribute addProperty PreviousPort "RC70_A3 (EK1122) : C"}
    {attribute addProperty SyncUnit "C70"}
    RC70_A5_EL1809 : EL1809_32157CFD;
    {attribute addProperty Name "RC70_A6 (EL1809)"}
    {attribute addProperty PreviousPort "RC70_A5 (EL1809) : B"}
    {attribute addProperty SyncUnit "C70"}
    RC70_A6_EL1809 : EL1809_32157CFD;
    {attribute addProperty Name "RC70_A7 (EL2809)"}
    {attribute addProperty PreviousPort "RC70_A6 (EL1809) : B"}
    {attribute addProperty SyncUnit "C70"}
    RC70_A7_EL2809 : EL2809_2B6483BD;
    {attribute addProperty Name "RC70_A8 (EL2809)"}
    {attribute addProperty PreviousPort "RC70_A7 (EL2809) : B"}
    {attribute addProperty SyncUnit "C70"}
    RC70_A8_EL2809 : EL2809_2B6483BD;
    {attribute addProperty Name "RC70_A9 (EL2809)"}
    {attribute addProperty PreviousPort "RC70_A8 (EL2809) : B"}
    {attribute addProperty SyncUnit "C70"}
    RC70_A9_EL2809 : EL2809_2B6483BD;
    {attribute addProperty Name "RC70_1_EndTerminal (EL9010)"}
    {attribute addProperty PreviousPort "RC70_A9 (EL2809) : B"}
    {attribute addProperty SyncUnit "default"}
    RC70_1_EndTerminal_EL9010 : EL9010_D29C2085;
END_STRUCT
END_TYPE

// ---- DUTs/IO/Topology/RC70_2_EK1100_D5DD9671.TcDUT
{attribute 'GeneratedUsingTerminal: EK1100-0000-0018'}
{attribute addProperty BoxType "EK1100-0000-0018"}
{attribute addProperty Id "RC70_B1_EL7041_1000EL7041_86DE63E743RC70_B2_EL7041_1000EL7041_86DE63E743RC70_C11_EL7041_1000EL7041_86DE63E743RC70_C12_EL7041_1000EL7041_86DE63E743RC70_C21_EL7041_1000EL7041_86DE63E743RC70_C22_EL7041_1000EL7041_86DE63E743RC70_2_EndTerminal_EL9010EL9010_D29C20850"}
{attribute addProperty CRC "3588068977"}
{attribute addProperty Size "258"}
{attribute addProperty Name "RC70_2 (EK1100)"}
TYPE RC70_2_EK1100_D5DD9671 EXTENDS EK1100_1FC0878B :
STRUCT
    {attribute addProperty Name "RC70_B1 (EL7041-1000)"}
    {attribute addProperty PreviousPort "RC70_2 (EK1100) : B"}
    {attribute addProperty SyncUnit "C70"}
    RC70_B1_EL7041_1000 : EL7041_86DE63E7;
    {attribute addProperty Name "RC70_B2 (EL7041-1000)"}
    {attribute addProperty PreviousPort "RC70_B1 (EL7041-1000) : B"}
    {attribute addProperty SyncUnit "C70"}
    RC70_B2_EL7041_1000 : EL7041_86DE63E7;
    {attribute addProperty Name "RC70_C11 (EL7041-1000)"}
    {attribute addProperty PreviousPort "RC70_B2 (EL7041-1000) : B"}
    {attribute addProperty SyncUnit "C70"}
    RC70_C11_EL7041_1000 : EL7041_86DE63E7;
    {attribute addProperty Name "RC70_C12 (EL7041-1000)"}
    {attribute addProperty PreviousPort "RC70_C11 (EL7041-1000) : B"}
    {attribute addProperty SyncUnit "C70"}
    RC70_C12_EL7041_1000 : EL7041_86DE63E7;
    {attribute addProperty Name "RC70_C21 (EL7041-1000)"}
    {attribute addProperty PreviousPort "RC70_C12 (EL7041-1000) : B"}
    {attribute addProperty SyncUnit "C70"}
    RC70_C21_EL7041_1000 : EL7041_86DE63E7;
    {attribute addProperty Name "RC70_C22 (EL7041-1000)"}
    {attribute addProperty PreviousPort "RC70_C21 (EL7041-1000) : B"}
    {attribute addProperty SyncUnit "C70"}
    RC70_C22_EL7041_1000 : EL7041_86DE63E7;
    {attribute addProperty Name "RC70_2_EndTerminal (EL9010)"}
    {attribute addProperty PreviousPort "RC70_C22 (EL7041-1000) : B"}
    {attribute addProperty SyncUnit "default"}
    RC70_2_EndTerminal_EL9010 : EL9010_D29C2085;
END_STRUCT
END_TYPE

// ---- DUTs/IO/Topology/RC80_A2_EK1122_C3467012.TcDUT
{attribute 'GeneratedUsingTerminal: EK1122-0000-0018'}
{attribute addProperty BoxType "EK1122-0000-0018"}
{attribute addProperty Id "RC80_VI_AES_D_BC_ECAT_xAES_B47A261080RC80_SAFETY_Flexi_Soft_EtherCAT_GatewayFlexi_Soft_EtherCAT_Gateway_DE394EDD5"}
{attribute addProperty CRC "3276173330"}
{attribute addProperty Size "85"}
{attribute addProperty Name "RC80_A2 (EK1122)"}
TYPE RC80_A2_EK1122_C3467012 EXTENDS EK1122_1FC0878B :
STRUCT
    {attribute addProperty Name "RC80_VI (AES-D-BC-ECAT)"}
    {attribute addProperty PreviousPort "RC80_A2 (EK1122) : D"}
    {attribute addProperty SyncUnit "C80"}
    RC80_VI_AES_D_BC_ECAT_x : AES_B47A2610;
    {attribute addProperty Name "RC80_SAFETY (Flexi Soft EtherCAT Gateway)"}
    {attribute addProperty PreviousPort "RC80_A2 (EK1122) : B"}
    {attribute addProperty SyncUnit "C80"}
    RC80_SAFETY_Flexi_Soft_EtherCAT_Gateway : Flexi_Soft_EtherCAT_Gateway_DE394EDD;
END_STRUCT
END_TYPE

// ---- DUTs/IO/Topology/RC80_EPP_EPP1322_0001_828B97C8.TcDUT
{attribute 'GeneratedUsingTerminal: EPP1322-0001-0017'}
{attribute addProperty BoxType "EPP1322-0001-0017"}
{attribute addProperty Id "RC80_AB1_EPP1008_0001EPP1008_78E8D3DD12RC80_AB2_EPP1008_0001EPP1008_78E8D3DD12RC80_AB6_EPP1008_0001EPP1008_78E8D3DD12RC80_AB3_EPP1008_0001EPP1008_78E8D3DD12RC80_AB4_EPP1008_0001EPP1008_78E8D3DD12RC80_AB7_EPP1008_0001EPP1008_78E8D3DD12RC80_AB9_EPP1008_0001EPP1008_78E8D3DD12RC80_AB10_EPP1008_0001EPP1008_78E8D3DD12RC80_AB8_EPP1008_0001EPP1008_78E8D3DD12RC80_AB5_EPP1008_0001EPP1008_78E8D3DD12"}
{attribute addProperty CRC "2190186440"}
{attribute addProperty Size "120"}
{attribute addProperty Name "RC80_EPP (EPP1322-0001)"}
TYPE RC80_EPP_EPP1322_0001_828B97C8 EXTENDS EPP1322_1FC0878B :
STRUCT
    {attribute addProperty Name "RC80_AB1 (EPP1008-0001)"}
    {attribute addProperty PreviousPort "RC80_EPP (EPP1322-0001) : D"}
    {attribute addProperty SyncUnit "C80"}
    RC80_AB1_EPP1008_0001 : EPP1008_78E8D3DD;
    {attribute addProperty Name "RC80_AB2 (EPP1008-0001)"}
    {attribute addProperty PreviousPort "RC80_AB1 (EPP1008-0001) : B"}
    {attribute addProperty SyncUnit "C80"}
    RC80_AB2_EPP1008_0001 : EPP1008_78E8D3DD;
    {attribute addProperty Name "RC80_AB6 (EPP1008-0001)"}
    {attribute addProperty PreviousPort "RC80_AB2 (EPP1008-0001) : B"}
    {attribute addProperty SyncUnit "C80"}
    RC80_AB6_EPP1008_0001 : EPP1008_78E8D3DD;
    {attribute addProperty Name "RC80_AB3 (EPP1008-0001)"}
    {attribute addProperty PreviousPort "RC80_AB6 (EPP1008-0001) : B"}
    {attribute addProperty SyncUnit "C80"}
    RC80_AB3_EPP1008_0001 : EPP1008_78E8D3DD;
    {attribute addProperty Name "RC80_AB4 (EPP1008-0001)"}
    {attribute addProperty PreviousPort "RC80_AB3 (EPP1008-0001) : B"}
    {attribute addProperty SyncUnit "C80"}
    RC80_AB4_EPP1008_0001 : EPP1008_78E8D3DD;
    {attribute addProperty Name "RC80_AB7 (EPP1008-0001)"}
    {attribute addProperty PreviousPort "RC80_EPP (EPP1322-0001) : B"}
    {attribute addProperty SyncUnit "C80"}
    RC80_AB7_EPP1008_0001 : EPP1008_78E8D3DD;
    {attribute addProperty Name "RC80_AB9 (EPP1008-0001)"}
    {attribute addProperty PreviousPort "RC80_AB7 (EPP1008-0001) : B"}
    {attribute addProperty SyncUnit "C80"}
    RC80_AB9_EPP1008_0001 : EPP1008_78E8D3DD;
    {attribute addProperty Name "RC80_AB10 (EPP1008-0001)"}
    {attribute addProperty PreviousPort "RC80_AB9 (EPP1008-0001) : B"}
    {attribute addProperty SyncUnit "C80"}
    RC80_AB10_EPP1008_0001 : EPP1008_78E8D3DD;
    {attribute addProperty Name "RC80_AB8 (EPP1008-0001)"}
    {attribute addProperty PreviousPort "RC80_AB10 (EPP1008-0001) : B"}
    {attribute addProperty SyncUnit "C80"}
    RC80_AB8_EPP1008_0001 : EPP1008_78E8D3DD;
    {attribute addProperty Name "RC80_AB5 (EPP1008-0001)"}
    {attribute addProperty PreviousPort "RC80_AB8 (EPP1008-0001) : B"}
    {attribute addProperty SyncUnit "C80"}
    RC80_AB5_EPP1008_0001 : EPP1008_78E8D3DD;
END_STRUCT
END_TYPE

// ---- DUTs/IO/Topology/RC80_A3_EK1122_B1484BA9.TcDUT
{attribute 'GeneratedUsingTerminal: EK1122-0000-0018'}
{attribute addProperty BoxType "EK1122-0000-0018"}
{attribute addProperty Id "RC80_EPP_EPP1322_0001RC80_EPP_EPP1322_0001_828B97C8120"}
{attribute addProperty CRC "2974305193"}
{attribute addProperty Size "120"}
{attribute addProperty Name "RC80_A3 (EK1122)"}
TYPE RC80_A3_EK1122_B1484BA9 EXTENDS EK1122_1FC0878B :
STRUCT
    {attribute addProperty Name "RC80_EPP (EPP1322-0001)"}
    {attribute addProperty PreviousPort "RC80_A3 (EK1122) : D"}
    {attribute addProperty SyncUnit "default"}
    RC80_EPP_EPP1322_0001 : RC80_EPP_EPP1322_0001_828B97C8;
END_STRUCT
END_TYPE

// ---- DUTs/IO/Topology/RC80_1_EK1100_5DD08FF5.TcDUT
{attribute 'GeneratedUsingTerminal: EK1100-0000-0018'}
{attribute addProperty BoxType "EK1100-0000-0018"}
{attribute addProperty Id "RC80_A2_EK1122RC80_A2_EK1122_C346701285RC80_A3_EK1122RC80_A3_EK1122_B1484BA9120RC80_A5_EL1809EL1809_32157CFD20RC80_A6_EL1809EL1809_32157CFD20RC80_A7_EL2809EL2809_2B6483BD19RC80_A8_EL2809EL2809_2B6483BD19RC80_A9_EL2809EL2809_2B6483BD19Term_796_EL9010EL9010_D29C20850"}
{attribute addProperty CRC "1573949429"}
{attribute addProperty Size "302"}
{attribute addProperty Name "RC80_1 (EK1100)"}
TYPE RC80_1_EK1100_5DD08FF5 EXTENDS EK1100_1FC0878B :
STRUCT
    {attribute addProperty Name "RC80_A2 (EK1122)"}
    {attribute addProperty PreviousPort "RC80_1 (EK1100) : B"}
    {attribute addProperty SyncUnit "default"}
    RC80_A2_EK1122 : RC80_A2_EK1122_C3467012;
    {attribute addProperty Name "RC80_A3 (EK1122)"}
    {attribute addProperty PreviousPort "RC80_A2 (EK1122) : C"}
    {attribute addProperty SyncUnit "default"}
    RC80_A3_EK1122 : RC80_A3_EK1122_B1484BA9;
    {attribute addProperty Name "RC80_A5 (EL1809)"}
    {attribute addProperty PreviousPort "RC80_A3 (EK1122) : C"}
    {attribute addProperty SyncUnit "C80"}
    RC80_A5_EL1809 : EL1809_32157CFD;
    {attribute addProperty Name "RC80_A6 (EL1809)"}
    {attribute addProperty PreviousPort "RC80_A5 (EL1809) : B"}
    {attribute addProperty SyncUnit "C80"}
    RC80_A6_EL1809 : EL1809_32157CFD;
    {attribute addProperty Name "RC80_A7 (EL2809)"}
    {attribute addProperty PreviousPort "RC80_A6 (EL1809) : B"}
    {attribute addProperty SyncUnit "C80"}
    RC80_A7_EL2809 : EL2809_2B6483BD;
    {attribute addProperty Name "RC80_A8 (EL2809)"}
    {attribute addProperty PreviousPort "RC80_A7 (EL2809) : B"}
    {attribute addProperty SyncUnit "C80"}
    RC80_A8_EL2809 : EL2809_2B6483BD;
    {attribute addProperty Name "RC80_A9 (EL2809)"}
    {attribute addProperty PreviousPort "RC80_A8 (EL2809) : B"}
    {attribute addProperty SyncUnit "C80"}
    RC80_A9_EL2809 : EL2809_2B6483BD;
    {attribute addProperty Name "Term 796 (EL9010)"}
    {attribute addProperty PreviousPort "RC80_A9 (EL2809) : B"}
    {attribute addProperty SyncUnit "default"}
    Term_796_EL9010 : EL9010_D29C2085;
END_STRUCT
END_TYPE

// ---- DUTs/IO/Topology/RC80_2_EK1100_DC1461B5.TcDUT
{attribute 'GeneratedUsingTerminal: EK1100-0000-0018'}
{attribute addProperty BoxType "EK1100-0000-0018"}
{attribute addProperty Id "RC80_B1_EL7041_1000EL7041_86DE63E743RC80_B2_EL7041_1000EL7041_86DE63E743RC80_C11_EL7041_1000EL7041_86DE63E743RC80_C12_EL7041_1000EL7041_86DE63E743RC80_C21_EL7041_1000EL7041_86DE63E743RC80_C22_EL7041_1000EL7041_86DE63E743Term_804_EL9010EL9010_D29C20850"}
{attribute addProperty CRC "3692323253"}
{attribute addProperty Size "258"}
{attribute addProperty Name "RC80_2 (EK1100)"}
TYPE RC80_2_EK1100_DC1461B5 EXTENDS EK1100_1FC0878B :
STRUCT
    {attribute addProperty Name "RC80_B1 (EL7041-1000)"}
    {attribute addProperty PreviousPort "RC80_2 (EK1100) : B"}
    {attribute addProperty SyncUnit "C80"}
    RC80_B1_EL7041_1000 : EL7041_86DE63E7;
    {attribute addProperty Name "RC80_B2 (EL7041-1000)"}
    {attribute addProperty PreviousPort "RC80_B1 (EL7041-1000) : B"}
    {attribute addProperty SyncUnit "C80"}
    RC80_B2_EL7041_1000 : EL7041_86DE63E7;
    {attribute addProperty Name "RC80_C11 (EL7041-1000)"}
    {attribute addProperty PreviousPort "RC80_B2 (EL7041-1000) : B"}
    {attribute addProperty SyncUnit "C80"}
    RC80_C11_EL7041_1000 : EL7041_86DE63E7;
    {attribute addProperty Name "RC80_C12 (EL7041-1000)"}
    {attribute addProperty PreviousPort "RC80_C11 (EL7041-1000) : B"}
    {attribute addProperty SyncUnit "C80"}
    RC80_C12_EL7041_1000 : EL7041_86DE63E7;
    {attribute addProperty Name "RC80_C21 (EL7041-1000)"}
    {attribute addProperty PreviousPort "RC80_C12 (EL7041-1000) : B"}
    {attribute addProperty SyncUnit "C80"}
    RC80_C21_EL7041_1000 : EL7041_86DE63E7;
    {attribute addProperty Name "RC80_C22 (EL7041-1000)"}
    {attribute addProperty PreviousPort "RC80_C21 (EL7041-1000) : B"}
    {attribute addProperty SyncUnit "C80"}
    RC80_C22_EL7041_1000 : EL7041_86DE63E7;
    {attribute addProperty Name "Term 804 (EL9010)"}
    {attribute addProperty PreviousPort "RC80_C22 (EL7041-1000) : B"}
    {attribute addProperty SyncUnit "default"}
    Term_804_EL9010 : EL9010_D29C2085;
END_STRUCT
END_TYPE

// ---- DUTs/IO/Topology/R8_A11_EK1122_3ED7E2A8.TcDUT
{attribute 'GeneratedUsingTerminal: EK1122-0000-0018'}
{attribute addProperty BoxType "EK1122-0000-0018"}
{attribute addProperty Id "RC70_1_EK1100RC70_1_EK1100_B905944A290RC70_2_EK1100RC70_2_EK1100_D5DD9671258RC80_1_EK1100RC80_1_EK1100_5DD08FF5302RC80_2_EK1100RC80_2_EK1100_DC1461B5258"}
{attribute addProperty CRC "1054335656"}
{attribute addProperty Size "1108"}
{attribute addProperty Name "R8_A11 (EK1122)"}
TYPE R8_A11_EK1122_3ED7E2A8 EXTENDS EK1122_1FC0878B :
STRUCT
    {attribute addProperty Name "RC70_1 (EK1100)"}
    {attribute addProperty PreviousPort "R8_A11 (EK1122) : D"}
    {attribute addProperty SyncUnit "default"}
    RC70_1_EK1100 : RC70_1_EK1100_B905944A;
    {attribute addProperty Name "RC70_2 (EK1100)"}
    {attribute addProperty PreviousPort "RC70_1 (EK1100) : C"}
    {attribute addProperty SyncUnit "default"}
    RC70_2_EK1100 : RC70_2_EK1100_D5DD9671;
    {attribute addProperty Name "RC80_1 (EK1100)"}
    {attribute addProperty PreviousPort "R8_A11 (EK1122) : B"}
    {attribute addProperty SyncUnit "default"}
    RC80_1_EK1100 : RC80_1_EK1100_5DD08FF5;
    {attribute addProperty Name "RC80_2 (EK1100)"}
    {attribute addProperty PreviousPort "RC80_1 (EK1100) : C"}
    {attribute addProperty SyncUnit "default"}
    RC80_2_EK1100 : RC80_2_EK1100_DC1461B5;
END_STRUCT
END_TYPE

// ---- DUTs/IO/Topology/RP10_A2_EK1122_55AC9C5A.TcDUT
{attribute 'GeneratedUsingTerminal: EK1122-0000-0018'}
{attribute addProperty BoxType "EK1122-0000-0018"}
{attribute addProperty Id "RP10_VI_AES_D_BC_ECAT_xAES_B47A261080RP10_SAFETY_Flexi_Soft_EtherCAT_GatewayFlexi_Soft_EtherCAT_Gateway_DE394EDD5RP10_AB0_EPP1322_0001EPP1322_1FC0878B2RP10_AB1_EPP1008_0001EPP1008_78E8D3DD12RP10_AB2_EPP1008_0001EPP1008_78E8D3DD12RP10_AB3_EPP1008_0001EPP1008_78E8D3DD12RP10_AB4_EPP1008_0001EPP1008_78E8D3DD12"}
{attribute addProperty CRC "1437375578"}
{attribute addProperty Size "135"}
{attribute addProperty Name "RP10_A2 (EK1122)"}
TYPE RP10_A2_EK1122_55AC9C5A EXTENDS EK1122_1FC0878B :
STRUCT
    {attribute addProperty Name "RP10-VI (AES-D-BC-ECAT)"}
    {attribute addProperty PreviousPort "RP10_A2 (EK1122) : D"}
    {attribute addProperty SyncUnit "P10"}
    RP10_VI_AES_D_BC_ECAT_x : AES_B47A2610;
    {attribute addProperty Name "RP10-SAFETY (Flexi Soft EtherCAT Gateway)"}
    {attribute addProperty PreviousPort "RP10_A2 (EK1122) : B"}
    {attribute addProperty SyncUnit "P10"}
    RP10_SAFETY_Flexi_Soft_EtherCAT_Gateway : Flexi_Soft_EtherCAT_Gateway_DE394EDD;
    {attribute addProperty Name "RP10-AB0 (EPP1322-0001)"}
    {attribute addProperty PreviousPort "RP10-SAFETY (Flexi Soft EtherCAT Gateway) : B"}
    {attribute addProperty SyncUnit "default"}
    RP10_AB0_EPP1322_0001 : EPP1322_1FC0878B;
    {attribute addProperty Name "RP10-AB1 (EPP1008-0001)"}
    {attribute addProperty PreviousPort "RP10-AB0 (EPP1322-0001) : C"}
    {attribute addProperty SyncUnit "P10"}
    RP10_AB1_EPP1008_0001 : EPP1008_78E8D3DD;
    {attribute addProperty Name "RP10-AB2 (EPP1008-0001)"}
    {attribute addProperty PreviousPort "RP10-AB1 (EPP1008-0001) : B"}
    {attribute addProperty SyncUnit "P10"}
    RP10_AB2_EPP1008_0001 : EPP1008_78E8D3DD;
    {attribute addProperty Name "RP10-AB3 (EPP1008-0001)"}
    {attribute addProperty PreviousPort "RP10-AB2 (EPP1008-0001) : B"}
    {attribute addProperty SyncUnit "P10"}
    RP10_AB3_EPP1008_0001 : EPP1008_78E8D3DD;
    {attribute addProperty Name "RP10-AB4 (EPP1008-0001)"}
    {attribute addProperty PreviousPort "RP10-AB3 (EPP1008-0001) : B"}
    {attribute addProperty SyncUnit "P10"}
    RP10_AB4_EPP1008_0001 : EPP1008_78E8D3DD;
END_STRUCT
END_TYPE

// ---- DUTs/IO/Topology/RP10_EK1100_26DB4001.TcDUT
{attribute 'GeneratedUsingTerminal: EK1100-0000-0018'}
{attribute addProperty BoxType "EK1100-0000-0018"}
{attribute addProperty Id "RP10_A2_EK1122RP10_A2_EK1122_55AC9C5A135RP10_A4_EL7041_1000EL7041_86DE63E743RP10_A5_EL7041_1000EL7041_86DE63E743RP10_A6_EL1809EL1809_32157CFD20RP10_A7_EL2809EL2809_2B6483BD19RP10_EndTerminal_EL9011EL9011_D65D3D320"}
{attribute addProperty CRC "651902977"}
{attribute addProperty Size "260"}
{attribute addProperty Name "RP10 (EK1100)"}
TYPE RP10_EK1100_26DB4001 EXTENDS EK1100_1FC0878B :
STRUCT
    {attribute addProperty Name "RP10_A2 (EK1122)"}
    {attribute addProperty PreviousPort "RP10 (EK1100) : B"}
    {attribute addProperty SyncUnit "default"}
    RP10_A2_EK1122 : RP10_A2_EK1122_55AC9C5A;
    {attribute addProperty Name "RP10_A4 (EL7041-1000)"}
    {attribute addProperty PreviousPort "RP10_A2 (EK1122) : C"}
    {attribute addProperty SyncUnit "P10"}
    RP10_A4_EL7041_1000 : EL7041_86DE63E7;
    {attribute addProperty Name "RP10_A5 (EL7041-1000)"}
    {attribute addProperty PreviousPort "RP10_A4 (EL7041-1000) : B"}
    {attribute addProperty SyncUnit "P10"}
    RP10_A5_EL7041_1000 : EL7041_86DE63E7;
    {attribute addProperty Name "RP10_A6 (EL1809)"}
    {attribute addProperty PreviousPort "RP10_A5 (EL7041-1000) : B"}
    {attribute addProperty SyncUnit "P10"}
    RP10_A6_EL1809 : EL1809_32157CFD;
    {attribute addProperty Name "RP10_A7 (EL2809)"}
    {attribute addProperty PreviousPort "RP10_A6 (EL1809) : B"}
    {attribute addProperty SyncUnit "P10"}
    RP10_A7_EL2809 : EL2809_2B6483BD;
    {attribute addProperty Name "RP10_EndTerminal (EL9011)"}
    {attribute addProperty PreviousPort "RP10_A7 (EL2809) : B"}
    {attribute addProperty SyncUnit "default"}
    RP10_EndTerminal_EL9011 : EL9011_D65D3D32;
END_STRUCT
END_TYPE

// ---- DUTs/IO/Topology/RP20_A2_EK1122_68D808EA.TcDUT
{attribute 'GeneratedUsingTerminal: EK1122-0000-0018'}
{attribute addProperty BoxType "EK1122-0000-0018"}
{attribute addProperty Id "RP20_VI_AES_D_BC_ECAT_xAES_B47A261080RP20_SAFETY_Flexi_Soft_EtherCAT_GatewayFlexi_Soft_EtherCAT_Gateway_DE394EDD5RP20_AB0_EPP1322_0001EPP1322_1FC0878B2RP20_AB1_EPP1008_0001EPP1008_78E8D3DD12RP20_AB2_EPP1008_0001EPP1008_78E8D3DD12RP20_AB3_EPP1008_0001EPP1008_78E8D3DD12RP20_AB4_EPP1008_0001EPP1008_78E8D3DD12"}
{attribute addProperty CRC "1758988522"}
{attribute addProperty Size "135"}
{attribute addProperty Name "RP20_A2 (EK1122)"}
TYPE RP20_A2_EK1122_68D808EA EXTENDS EK1122_1FC0878B :
STRUCT
    {attribute addProperty Name "RP20-VI (AES-D-BC-ECAT)"}
    {attribute addProperty PreviousPort "RP20_A2 (EK1122) : D"}
    {attribute addProperty SyncUnit "P20"}
    RP20_VI_AES_D_BC_ECAT_x : AES_B47A2610;
    {attribute addProperty Name "RP20-SAFETY (Flexi Soft EtherCAT Gateway)"}
    {attribute addProperty PreviousPort "RP20_A2 (EK1122) : B"}
    {attribute addProperty SyncUnit "P20"}
    RP20_SAFETY_Flexi_Soft_EtherCAT_Gateway : Flexi_Soft_EtherCAT_Gateway_DE394EDD;
    {attribute addProperty Name "RP20-AB0 (EPP1322-0001)"}
    {attribute addProperty PreviousPort "RP20-SAFETY (Flexi Soft EtherCAT Gateway) : B"}
    {attribute addProperty SyncUnit "default"}
    RP20_AB0_EPP1322_0001 : EPP1322_1FC0878B;
    {attribute addProperty Name "RP20-AB1 (EPP1008-0001)"}
    {attribute addProperty PreviousPort "RP20-AB0 (EPP1322-0001) : C"}
    {attribute addProperty SyncUnit "P20"}
    RP20_AB1_EPP1008_0001 : EPP1008_78E8D3DD;
    {attribute addProperty Name "RP20-AB2 (EPP1008-0001)"}
    {attribute addProperty PreviousPort "RP20-AB1 (EPP1008-0001) : B"}
    {attribute addProperty SyncUnit "P20"}
    RP20_AB2_EPP1008_0001 : EPP1008_78E8D3DD;
    {attribute addProperty Name "RP20-AB3 (EPP1008-0001)"}
    {attribute addProperty PreviousPort "RP20-AB2 (EPP1008-0001) : B"}
    {attribute addProperty SyncUnit "P20"}
    RP20_AB3_EPP1008_0001 : EPP1008_78E8D3DD;
    {attribute addProperty Name "RP20-AB4 (EPP1008-0001)"}
    {attribute addProperty PreviousPort "RP20-AB3 (EPP1008-0001) : B"}
    {attribute addProperty SyncUnit "P20"}
    RP20_AB4_EPP1008_0001 : EPP1008_78E8D3DD;
END_STRUCT
END_TYPE

// ---- DUTs/IO/Topology/RP20_EK1100_7A23D5FF.TcDUT
{attribute 'GeneratedUsingTerminal: EK1100-0000-0018'}
{attribute addProperty BoxType "EK1100-0000-0018"}
{attribute addProperty Id "RP20_A2_EK1122RP20_A2_EK1122_68D808EA135RP20_A4_EL7041_1000EL7041_86DE63E743RP20_A5_EL7041_1000EL7041_86DE63E743RP20_A6_EL1809EL1809_32157CFD20RP20_A7_EL2809EL2809_2B6483BD19RP20_EndTerminal_EL9011EL9011_D65D3D320"}
{attribute addProperty CRC "2049168895"}
{attribute addProperty Size "260"}
{attribute addProperty Name "RP20 (EK1100)"}
TYPE RP20_EK1100_7A23D5FF EXTENDS EK1100_1FC0878B :
STRUCT
    {attribute addProperty Name "RP20_A2 (EK1122)"}
    {attribute addProperty PreviousPort "RP20 (EK1100) : B"}
    {attribute addProperty SyncUnit "default"}
    RP20_A2_EK1122 : RP20_A2_EK1122_68D808EA;
    {attribute addProperty Name "RP20_A4 (EL7041-1000)"}
    {attribute addProperty PreviousPort "RP20_A2 (EK1122) : C"}
    {attribute addProperty SyncUnit "P20"}
    RP20_A4_EL7041_1000 : EL7041_86DE63E7;
    {attribute addProperty Name "RP20_A5 (EL7041-1000)"}
    {attribute addProperty PreviousPort "RP20_A4 (EL7041-1000) : B"}
    {attribute addProperty SyncUnit "P20"}
    RP20_A5_EL7041_1000 : EL7041_86DE63E7;
    {attribute addProperty Name "RP20_A6 (EL1809)"}
    {attribute addProperty PreviousPort "RP20_A5 (EL7041-1000) : B"}
    {attribute addProperty SyncUnit "P20"}
    RP20_A6_EL1809 : EL1809_32157CFD;
    {attribute addProperty Name "RP20_A7 (EL2809)"}
    {attribute addProperty PreviousPort "RP20_A6 (EL1809) : B"}
    {attribute addProperty SyncUnit "P20"}
    RP20_A7_EL2809 : EL2809_2B6483BD;
    {attribute addProperty Name "RP20_EndTerminal (EL9011)"}
    {attribute addProperty PreviousPort "RP20_A7 (EL2809) : B"}
    {attribute addProperty SyncUnit "default"}
    RP20_EndTerminal_EL9011 : EL9011_D65D3D32;
END_STRUCT
END_TYPE

// ---- DUTs/IO/Topology/R8_A12_EK1122_5B843125.TcDUT
{attribute 'GeneratedUsingTerminal: EK1122-0000-0018'}
{attribute addProperty BoxType "EK1122-0000-0018"}
{attribute addProperty Id "RP10_EK1100RP10_EK1100_26DB4001260RP20_EK1100RP20_EK1100_7A23D5FF260"}
{attribute addProperty CRC "1535389989"}
{attribute addProperty Size "520"}
{attribute addProperty Name "R8_A12 (EK1122)"}
TYPE R8_A12_EK1122_5B843125 EXTENDS EK1122_1FC0878B :
STRUCT
    {attribute addProperty Name "RP10 (EK1100)"}
    {attribute addProperty PreviousPort "R8_A12 (EK1122) : D"}
    {attribute addProperty SyncUnit "default"}
    RP10_EK1100 : RP10_EK1100_26DB4001;
    {attribute addProperty Name "RP20 (EK1100)"}
    {attribute addProperty PreviousPort "R8_A12 (EK1122) : B"}
    {attribute addProperty SyncUnit "default"}
    RP20_EK1100 : RP20_EK1100_7A23D5FF;
END_STRUCT
END_TYPE

// ---- DUTs/IO/Topology/RP30_A2_EK1122_C3CC9CB4.TcDUT
{attribute 'GeneratedUsingTerminal: EK1122-0000-0018'}
{attribute addProperty BoxType "EK1122-0000-0018"}
{attribute addProperty Id "RP30_VI_AES_D_BC_ECAT_xAES_A3B0707168RP30_SAFETY_Flexi_Soft_EtherCAT_GatewayFlexi_Soft_EtherCAT_Gateway_DE394EDD5RP30_AB0_EPP1322_0001EPP1322_1FC0878B2RP30_AB1_EPP1008_0001EPP1008_78E8D3DD12RP30_AB2_EPP1008_0001EPP1008_78E8D3DD12RP30_AB3_EPP1008_0001EPP1008_78E8D3DD12RP30_AB4_EPP1008_0001EPP1008_78E8D3DD12"}
{attribute addProperty CRC "3284966580"}
{attribute addProperty Size "123"}
{attribute addProperty Name "RP30_A2 (EK1122)"}
TYPE RP30_A2_EK1122_C3CC9CB4 EXTENDS EK1122_1FC0878B :
STRUCT
    {attribute addProperty Name "RP30-VI (AES-D-BC-ECAT)"}
    {attribute addProperty PreviousPort "RP30_A2 (EK1122) : D"}
    {attribute addProperty SyncUnit "P30"}
    RP30_VI_AES_D_BC_ECAT_x : AES_A3B07071;
    {attribute addProperty Name "RP30-SAFETY (Flexi Soft EtherCAT Gateway)"}
    {attribute addProperty PreviousPort "RP30_A2 (EK1122) : B"}
    {attribute addProperty SyncUnit "P30"}
    RP30_SAFETY_Flexi_Soft_EtherCAT_Gateway : Flexi_Soft_EtherCAT_Gateway_DE394EDD;
    {attribute addProperty Name "RP30-AB0 (EPP1322-0001)"}
    {attribute addProperty PreviousPort "RP30-SAFETY (Flexi Soft EtherCAT Gateway) : B"}
    {attribute addProperty SyncUnit "default"}
    RP30_AB0_EPP1322_0001 : EPP1322_1FC0878B;
    {attribute addProperty Name "RP30-AB1 (EPP1008-0001)"}
    {attribute addProperty PreviousPort "RP30-AB0 (EPP1322-0001) : C"}
    {attribute addProperty SyncUnit "P30"}
    RP30_AB1_EPP1008_0001 : EPP1008_78E8D3DD;
    {attribute addProperty Name "RP30-AB2 (EPP1008-0001)"}
    {attribute addProperty PreviousPort "RP30-AB1 (EPP1008-0001) : B"}
    {attribute addProperty SyncUnit "P30"}
    RP30_AB2_EPP1008_0001 : EPP1008_78E8D3DD;
    {attribute addProperty Name "RP30-AB3 (EPP1008-0001)"}
    {attribute addProperty PreviousPort "RP30-AB2 (EPP1008-0001) : B"}
    {attribute addProperty SyncUnit "P30"}
    RP30_AB3_EPP1008_0001 : EPP1008_78E8D3DD;
    {attribute addProperty Name "RP30-AB4 (EPP1008-0001)"}
    {attribute addProperty PreviousPort "RP30-AB3 (EPP1008-0001) : B"}
    {attribute addProperty SyncUnit "P30"}
    RP30_AB4_EPP1008_0001 : EPP1008_78E8D3DD;
END_STRUCT
END_TYPE

// ---- DUTs/IO/Topology/RP30_EK1100_66AE6AB6.TcDUT
{attribute 'GeneratedUsingTerminal: EK1100-0000-0018'}
{attribute addProperty BoxType "EK1100-0000-0018"}
{attribute addProperty Id "RP30_A2_EK1122RP30_A2_EK1122_C3CC9CB4123RP30_A4_EL7041_1000EL7041_86DE63E743RP30_A5_EL7041_1000EL7041_86DE63E743RP30_A6_EL1809EL1809_32157CFD20RP30_A7_EL2809EL2809_2B6483BD19RP30_EndTerminal_EL9010EL9010_D29C20850"}
{attribute addProperty CRC "1722706614"}
{attribute addProperty Size "248"}
{attribute addProperty Name "RP30 (EK1100)"}
TYPE RP30_EK1100_66AE6AB6 EXTENDS EK1100_1FC0878B :
STRUCT
    {attribute addProperty Name "RP30_A2 (EK1122)"}
    {attribute addProperty PreviousPort "RP30 (EK1100) : B"}
    {attribute addProperty SyncUnit "default"}
    RP30_A2_EK1122 : RP30_A2_EK1122_C3CC9CB4;
    {attribute addProperty Name "RP30_A4 (EL7041-1000)"}
    {attribute addProperty PreviousPort "RP30_A2 (EK1122) : C"}
    {attribute addProperty SyncUnit "P30"}
    RP30_A4_EL7041_1000 : EL7041_86DE63E7;
    {attribute addProperty Name "RP30_A5 (EL7041-1000)"}
    {attribute addProperty PreviousPort "RP30_A4 (EL7041-1000) : B"}
    {attribute addProperty SyncUnit "P30"}
    RP30_A5_EL7041_1000 : EL7041_86DE63E7;
    {attribute addProperty Name "RP30_A6 (EL1809)"}
    {attribute addProperty PreviousPort "RP30_A5 (EL7041-1000) : B"}
    {attribute addProperty SyncUnit "P30"}
    RP30_A6_EL1809 : EL1809_32157CFD;
    {attribute addProperty Name "RP30_A7 (EL2809)"}
    {attribute addProperty PreviousPort "RP30_A6 (EL1809) : B"}
    {attribute addProperty SyncUnit "P30"}
    RP30_A7_EL2809 : EL2809_2B6483BD;
    {attribute addProperty Name "RP30_EndTerminal (EL9010)"}
    {attribute addProperty PreviousPort "RP30_A7 (EL2809) : B"}
    {attribute addProperty SyncUnit "default"}
    RP30_EndTerminal_EL9010 : EL9010_D29C2085;
END_STRUCT
END_TYPE

// ---- DUTs/IO/Topology/R8_A13_EK1122_C6957FFB.TcDUT
{attribute 'GeneratedUsingTerminal: EK1122-0000-0018'}
{attribute addProperty BoxType "EK1122-0000-0018"}
{attribute addProperty Id "RP30_EK1100RP30_EK1100_66AE6AB6248"}
{attribute addProperty CRC "3331686395"}
{attribute addProperty Size "248"}
{attribute addProperty Name "R8_A13 (EK1122)"}
TYPE R8_A13_EK1122_C6957FFB EXTENDS EK1122_1FC0878B :
STRUCT
    {attribute addProperty Name "RP30 (EK1100)"}
    {attribute addProperty PreviousPort "R8_A13 (EK1122) : D"}
    {attribute addProperty SyncUnit "default"}
    RP30_EK1100 : RP30_EK1100_66AE6AB6;
END_STRUCT
END_TYPE

// ---- DUTs/IO/Topology/R8_EK1100_9C7B3B67.TcDUT
{attribute 'GeneratedUsingTerminal: EK1100-0000-0018'}
{attribute addProperty BoxType "EK1100-0000-0018"}
{attribute addProperty Id "R8_A2_EK1122R8_A2_EK1122_E74C4B62290R8_A3_EK1122R8_A3_EK1122_71CA94BA136R8_A5_EL1809EL1809_32157CFD20R8_A6_EL2809EL2809_2B6483BD19R8_A7_EL2809EL2809_2B6483BD19R8_A8_EK1122R8_A8_EK1122_2533F93A1096R8_A9_EK1122R8_A9_EK1122_3EDD87521096R8_A10_EK1122R8_A10_EK1122_484442E01096R8_A11_EK1122R8_A11_EK1122_3ED7E2A81108R8_A12_EK1122R8_A12_EK1122_5B843125520R8_A13_EK1122R8_A13_EK1122_C6957FFB248R8_Endterminal_EL9010EL9010_D29C20850"}
{attribute addProperty CRC "2625321831"}
{attribute addProperty Size "5648"}
{attribute addProperty Name "R8 (EK1100)"}
TYPE R8_EK1100_9C7B3B67 EXTENDS EK1100_1FC0878B :
STRUCT
    {attribute addProperty Name "R8_A2 (EK1122)"}
    {attribute addProperty PreviousPort "R8 (EK1100) : B"}
    {attribute addProperty SyncUnit "default"}
    R8_A2_EK1122 : R8_A2_EK1122_E74C4B62;
    {attribute addProperty Name "R8_A3 (EK1122)"}
    {attribute addProperty PreviousPort "R8_A2 (EK1122) : C"}
    {attribute addProperty SyncUnit "default"}
    R8_A3_EK1122 : R8_A3_EK1122_71CA94BA;
    {attribute addProperty Name "R8_A5 (EL1809)"}
    {attribute addProperty PreviousPort "R8_A3 (EK1122) : C"}
    {attribute addProperty SyncUnit "default"}
    R8_A5_EL1809 : EL1809_32157CFD;
    {attribute addProperty Name "R8_A6 (EL2809)"}
    {attribute addProperty PreviousPort "R8_A5 (EL1809) : B"}
    {attribute addProperty SyncUnit "default"}
    R8_A6_EL2809 : EL2809_2B6483BD;
    {attribute addProperty Name "R8_A7 (EL2809)"}
    {attribute addProperty PreviousPort "R8_A6 (EL2809) : B"}
    {attribute addProperty SyncUnit "default"}
    R8_A7_EL2809 : EL2809_2B6483BD;
    {attribute addProperty Name "R8_A8 (EK1122)"}
    {attribute addProperty PreviousPort "R8_A7 (EL2809) : B"}
    {attribute addProperty SyncUnit "default"}
    R8_A8_EK1122 : R8_A8_EK1122_2533F93A;
    {attribute addProperty Name "R8_A9 (EK1122)"}
    {attribute addProperty PreviousPort "R8_A8 (EK1122) : C"}
    {attribute addProperty SyncUnit "default"}
    R8_A9_EK1122 : R8_A9_EK1122_3EDD8752;
    {attribute addProperty Name "R8_A10 (EK1122)"}
    {attribute addProperty PreviousPort "R8_A9 (EK1122) : C"}
    {attribute addProperty SyncUnit "default"}
    R8_A10_EK1122 : R8_A10_EK1122_484442E0;
    {attribute addProperty Name "R8_A11 (EK1122)"}
    {attribute addProperty PreviousPort "R8_A10 (EK1122) : C"}
    {attribute addProperty SyncUnit "default"}
    R8_A11_EK1122 : R8_A11_EK1122_3ED7E2A8;
    {attribute addProperty Name "R8_A12 (EK1122)"}
    {attribute addProperty PreviousPort "R8_A11 (EK1122) : C"}
    {attribute addProperty SyncUnit "default"}
    R8_A12_EK1122 : R8_A12_EK1122_5B843125;
    {attribute addProperty Name "R8_A13 (EK1122)"}
    {attribute addProperty PreviousPort "R8_A12 (EK1122) : C"}
    {attribute addProperty SyncUnit "default"}
    R8_A13_EK1122 : R8_A13_EK1122_C6957FFB;
    {attribute addProperty Name "R8_Endterminal (EL9010)"}
    {attribute addProperty PreviousPort "R8_A13 (EK1122) : C"}
    {attribute addProperty SyncUnit "default"}
    R8_Endterminal_EL9010 : EL9010_D29C2085;
END_STRUCT
END_TYPE

// ---- DUTs/IO/Topology/R9_AB0_EPP1322_0001_BD7A28FA.TcDUT
{attribute 'GeneratedUsingTerminal: EPP1322-0001-0017'}
{attribute addProperty BoxType "EPP1322-0001-0017"}
{attribute addProperty Id "R9_AB1_EPP1008_0001EPP1008_78E8D3DD12R9_AB2_EPP1008_0001EPP1008_78E8D3DD12R9_AB3_EPP1008_0001EPP1008_78E8D3DD12R9_AB4_EPP1008_0001EPP1008_78E8D3DD12"}
{attribute addProperty CRC "3178899706"}
{attribute addProperty Size "48"}
{attribute addProperty Name "R9_AB0 (EPP1322-0001)"}
TYPE R9_AB0_EPP1322_0001_BD7A28FA EXTENDS EPP1322_1FC0878B :
STRUCT
    {attribute addProperty Name "R9_AB1 (EPP1008-0001)"}
    {attribute addProperty PreviousPort "R9_AB0 (EPP1322-0001) : D"}
    {attribute addProperty SyncUnit "default"}
    R9_AB1_EPP1008_0001 : EPP1008_78E8D3DD;
    {attribute addProperty Name "R9_AB2 (EPP1008-0001)"}
    {attribute addProperty PreviousPort "R9_AB1 (EPP1008-0001) : B"}
    {attribute addProperty SyncUnit "default"}
    R9_AB2_EPP1008_0001 : EPP1008_78E8D3DD;
    {attribute addProperty Name "R9_AB3 (EPP1008-0001)"}
    {attribute addProperty PreviousPort "R9_AB2 (EPP1008-0001) : B"}
    {attribute addProperty SyncUnit "default"}
    R9_AB3_EPP1008_0001 : EPP1008_78E8D3DD;
    {attribute addProperty Name "R9_AB4 (EPP1008-0001)"}
    {attribute addProperty PreviousPort "R9_AB3 (EPP1008-0001) : B"}
    {attribute addProperty SyncUnit "default"}
    R9_AB4_EPP1008_0001 : EPP1008_78E8D3DD;
END_STRUCT
END_TYPE

// ---- DUTs/IO/Topology/R9_A2_EK1122_81F50509.TcDUT
{attribute 'GeneratedUsingTerminal: EK1122-0000-0018'}
{attribute addProperty BoxType "EK1122-0000-0018"}
{attribute addProperty Id "R9_AB0_EPP1322_0001R9_AB0_EPP1322_0001_BD7A28FA48R9_SAFETY_Flexi_Soft_EtherCAT_GatewayFlexi_Soft_EtherCAT_Gateway_DE394EDD5"}
{attribute addProperty CRC "2180318473"}
{attribute addProperty Size "53"}
{attribute addProperty Name "R9_A2 (EK1122)"}
TYPE R9_A2_EK1122_81F50509 EXTENDS EK1122_1FC0878B :
STRUCT
    {attribute addProperty Name "R9_AB0 (EPP1322-0001)"}
    {attribute addProperty PreviousPort "R9_A2 (EK1122) : D"}
    {attribute addProperty SyncUnit "default"}
    R9_AB0_EPP1322_0001 : R9_AB0_EPP1322_0001_BD7A28FA;
    {attribute addProperty Name "R9_SAFETY (Flexi Soft EtherCAT Gateway)"}
    {attribute addProperty PreviousPort "R9_A2 (EK1122) : B"}
    {attribute addProperty SyncUnit "default"}
    R9_SAFETY_Flexi_Soft_EtherCAT_Gateway : Flexi_Soft_EtherCAT_Gateway_DE394EDD;
END_STRUCT
END_TYPE

// ---- DUTs/IO/Topology/R9_A3_EK1122_C18C26F5.TcDUT
{attribute 'GeneratedUsingTerminal: EK1122-0000-0018'}
{attribute addProperty BoxType "EK1122-0000-0018"}
{attribute addProperty Id "R9_SERVO_IndraDrive_MPB20IndraDrive_MPB20_C66205C325"}
{attribute addProperty CRC "3247187701"}
{attribute addProperty Size "25"}
{attribute addProperty Name "R9_A3 (EK1122)"}
TYPE R9_A3_EK1122_C18C26F5 EXTENDS EK1122_1FC0878B :
STRUCT
    {attribute addProperty Name "R9_SERVO (IndraDrive MPB20)"}
    {attribute addProperty PreviousPort "R9_A3 (EK1122) : D"}
    {attribute addProperty SyncUnit "default"}
    R9_SERVO_IndraDrive_MPB20 : IndraDrive_MPB20_C66205C3;
END_STRUCT
END_TYPE

// ---- DUTs/IO/Topology/R9_EK1100_484053C0.TcDUT
{attribute 'GeneratedUsingTerminal: EK1100-0000-0018'}
{attribute addProperty BoxType "EK1100-0000-0018"}
{attribute addProperty Id "R9_A2_EK1122R9_A2_EK1122_81F5050953R9_A3_EK1122R9_A3_EK1122_C18C26F525R9_A5_EL1809EL1809_32157CFD20R9_A6_EL2809EL2809_2B6483BD19R9_A7_EL2809EL2809_2B6483BD19R9_EndTerminal_EL9011EL9011_D65D3D320"}
{attribute addProperty CRC "1212175296"}
{attribute addProperty Size "136"}
{attribute addProperty Name "R9 (EK1100)"}
TYPE R9_EK1100_484053C0 EXTENDS EK1100_1FC0878B :
STRUCT
    {attribute addProperty Name "R9_A2 (EK1122)"}
    {attribute addProperty PreviousPort "R9 (EK1100) : B"}
    {attribute addProperty SyncUnit "default"}
    R9_A2_EK1122 : R9_A2_EK1122_81F50509;
    {attribute addProperty Name "R9_A3 (EK1122)"}
    {attribute addProperty PreviousPort "R9_A2 (EK1122) : C"}
    {attribute addProperty SyncUnit "default"}
    R9_A3_EK1122 : R9_A3_EK1122_C18C26F5;
    {attribute addProperty Name "R9_A5 (EL1809)"}
    {attribute addProperty PreviousPort "R9_A3 (EK1122) : C"}
    {attribute addProperty SyncUnit "default"}
    R9_A5_EL1809 : EL1809_32157CFD;
    {attribute addProperty Name "R9_A6 (EL2809)"}
    {attribute addProperty PreviousPort "R9_A5 (EL1809) : B"}
    {attribute addProperty SyncUnit "default"}
    R9_A6_EL2809 : EL2809_2B6483BD;
    {attribute addProperty Name "R9_A7 (EL2809)"}
    {attribute addProperty PreviousPort "R9_A6 (EL2809) : B"}
    {attribute addProperty SyncUnit "default"}
    R9_A7_EL2809 : EL2809_2B6483BD;
    {attribute addProperty Name "R9_EndTerminal (EL9011)"}
    {attribute addProperty PreviousPort "R9_A7 (EL2809) : B"}
    {attribute addProperty SyncUnit "default"}
    R9_EndTerminal_EL9011 : EL9011_D65D3D32;
END_STRUCT
END_TYPE

// ---- DUTs/IO/Topology/R10_A2_EK1122_75D61001.TcDUT
{attribute 'GeneratedUsingTerminal: EK1122-0000-0018'}
{attribute addProperty BoxType "EK1122-0000-0018"}
{attribute addProperty Id "R10_VI11_AES_D_BC_ECAT_xAES_B47A261080R10_VI12_AES_D_BC_ECAT_xAES_B47A261080R10_SAFETY_Flexi_Soft_EtherCAT_GatewayFlexi_Soft_EtherCAT_Gateway_DE394EDD5"}
{attribute addProperty CRC "1976963073"}
{attribute addProperty Size "165"}
{attribute addProperty Name "R10_A2 (EK1122)"}
TYPE R10_A2_EK1122_75D61001 EXTENDS EK1122_1FC0878B :
STRUCT
    {attribute addProperty Name "R10-VI11 (AES-D-BC-ECAT)"}
    {attribute addProperty PreviousPort "R10_A2 (EK1122) : D"}
    {attribute addProperty SyncUnit "R10"}
    R10_VI11_AES_D_BC_ECAT_x : AES_B47A2610;
    {attribute addProperty Name "R10-VI12 (AES-D-BC-ECAT)"}
    {attribute addProperty PreviousPort "R10-VI11 (AES-D-BC-ECAT) : B"}
    {attribute addProperty SyncUnit "R10"}
    R10_VI12_AES_D_BC_ECAT_x : AES_B47A2610;
    {attribute addProperty Name "R10_SAFETY (Flexi Soft EtherCAT Gateway)"}
    {attribute addProperty PreviousPort "R10_A2 (EK1122) : B"}
    {attribute addProperty SyncUnit "R10"}
    R10_SAFETY_Flexi_Soft_EtherCAT_Gateway : Flexi_Soft_EtherCAT_Gateway_DE394EDD;
END_STRUCT
END_TYPE

// ---- DUTs/IO/Topology/R10_AB01_EPP1332_0001_D97A7767.TcDUT
{attribute 'GeneratedUsingTerminal: EPP1332-0001-0017'}
{attribute addProperty BoxType "EPP1332-0001-0017"}
{attribute addProperty Id "R10_ABT8_EPP1008_0001EPP1008_78E8D3DD12R10_ABT9_EPP1008_0001EPP1008_78E8D3DD12R10_ABT10_EPP1008_0001EPP1008_78E8D3DD12R10_ABT11_EPP1008_0001EPP1008_78E8D3DD12R10_ABT12_EPP1008_0001EPP1008_78E8D3DD12"}
{attribute addProperty CRC "3648681831"}
{attribute addProperty Size "60"}
{attribute addProperty Name "R10-AB01 (EPP1332-0001)"}
TYPE R10_AB01_EPP1332_0001_D97A7767 EXTENDS EPP1332_1FC0878B :
STRUCT
    {attribute addProperty Name "R10-ABT8 (EPP1008-0001)"}
    {attribute addProperty PreviousPort "R10-AB01 (EPP1332-0001) : D"}
    {attribute addProperty SyncUnit "R10"}
    R10_ABT8_EPP1008_0001 : EPP1008_78E8D3DD;
    {attribute addProperty Name "R10-ABT9 (EPP1008-0001)"}
    {attribute addProperty PreviousPort "R10-ABT8 (EPP1008-0001) : B"}
    {attribute addProperty SyncUnit "R10"}
    R10_ABT9_EPP1008_0001 : EPP1008_78E8D3DD;
    {attribute addProperty Name "R10-ABT10 (EPP1008-0001)"}
    {attribute addProperty PreviousPort "R10-ABT9 (EPP1008-0001) : B"}
    {attribute addProperty SyncUnit "R10"}
    R10_ABT10_EPP1008_0001 : EPP1008_78E8D3DD;
    {attribute addProperty Name "R10-ABT11 (EPP1008-0001)"}
    {attribute addProperty PreviousPort "R10-ABT10 (EPP1008-0001) : B"}
    {attribute addProperty SyncUnit "R10"}
    R10_ABT11_EPP1008_0001 : EPP1008_78E8D3DD;
    {attribute addProperty Name "R10-ABT12 (EPP1008-0001)"}
    {attribute addProperty PreviousPort "R10-ABT11 (EPP1008-0001) : B"}
    {attribute addProperty SyncUnit "R10"}
    R10_ABT12_EPP1008_0001 : EPP1008_78E8D3DD;
END_STRUCT
END_TYPE

// ---- DUTs/IO/Topology/R10_AB00_EPP1322_0001_481BC624.TcDUT
{attribute 'GeneratedUsingTerminal: EPP1322-0001-0017'}
{attribute addProperty BoxType "EPP1322-0001-0017"}
{attribute addProperty Id "R10_AB9_EPP1008_0001EPP1008_78E8D3DD12R10_AB10_EPP1008_0001EPP1008_78E8D3DD12R10_AB01_EPP1332_0001R10_AB01_EPP1332_0001_D97A776760R10_ABT7_EPP1008_0001EPP1008_78E8D3DD12R10_ABT6_EPP1008_0001EPP1008_78E8D3DD12R10_ABT5_EPP1008_0001EPP1008_78E8D3DD12R10_ABT4_EPP1008_0001EPP1008_78E8D3DD12R10_ABT3_EPP1008_0001EPP1008_78E8D3DD12R10_ABT2_EPP1008_0001EPP1008_78E8D3DD12R10_ABT1_EPP1008_0001EPP1008_78E8D3DD12"}
{attribute addProperty CRC "1209779748"}
{attribute addProperty Size "168"}
{attribute addProperty Name "R10-AB00 (EPP1322-0001)"}
TYPE R10_AB00_EPP1322_0001_481BC624 EXTENDS EPP1322_1FC0878B :
STRUCT
    {attribute addProperty Name "R10-AB9 (EPP1008-0001)"}
    {attribute addProperty PreviousPort "R10-AB00 (EPP1322-0001) : D"}
    {attribute addProperty SyncUnit "R10"}
    R10_AB9_EPP1008_0001 : EPP1008_78E8D3DD;
    {attribute addProperty Name "R10-AB10 (EPP1008-0001)"}
    {attribute addProperty PreviousPort "R10-AB9 (EPP1008-0001) : B"}
    {attribute addProperty SyncUnit "R10"}
    R10_AB10_EPP1008_0001 : EPP1008_78E8D3DD;
    {attribute addProperty Name "R10-AB01 (EPP1332-0001)"}
    {attribute addProperty PreviousPort "R10-AB00 (EPP1322-0001) : B"}
    {attribute addProperty SyncUnit "default"}
    R10_AB01_EPP1332_0001 : R10_AB01_EPP1332_0001_D97A7767;
    {attribute addProperty Name "R10-ABT7 (EPP1008-0001)"}
    {attribute addProperty PreviousPort "R10-AB01 (EPP1332-0001) : C"}
    {attribute addProperty SyncUnit "R10"}
    R10_ABT7_EPP1008_0001 : EPP1008_78E8D3DD;
    {attribute addProperty Name "R10-ABT6 (EPP1008-0001)"}
    {attribute addProperty PreviousPort "R10-ABT7 (EPP1008-0001) : B"}
    {attribute addProperty SyncUnit "R10"}
    R10_ABT6_EPP1008_0001 : EPP1008_78E8D3DD;
    {attribute addProperty Name "R10-ABT5 (EPP1008-0001)"}
    {attribute addProperty PreviousPort "R10-ABT6 (EPP1008-0001) : B"}
    {attribute addProperty SyncUnit "R10"}
    R10_ABT5_EPP1008_0001 : EPP1008_78E8D3DD;
    {attribute addProperty Name "R10-ABT4 (EPP1008-0001)"}
    {attribute addProperty PreviousPort "R10-ABT5 (EPP1008-0001) : B"}
    {attribute addProperty SyncUnit "R10"}
    R10_ABT4_EPP1008_0001 : EPP1008_78E8D3DD;
    {attribute addProperty Name "R10-ABT3 (EPP1008-0001)"}
    {attribute addProperty PreviousPort "R10-ABT4 (EPP1008-0001) : B"}
    {attribute addProperty SyncUnit "R10"}
    R10_ABT3_EPP1008_0001 : EPP1008_78E8D3DD;
    {attribute addProperty Name "R10-ABT2 (EPP1008-0001)"}
    {attribute addProperty PreviousPort "R10-ABT3 (EPP1008-0001) : B"}
    {attribute addProperty SyncUnit "R10"}
    R10_ABT2_EPP1008_0001 : EPP1008_78E8D3DD;
    {attribute addProperty Name "R10-ABT1 (EPP1008-0001)"}
    {attribute addProperty PreviousPort "R10-ABT2 (EPP1008-0001) : B"}
    {attribute addProperty SyncUnit "R10"}
    R10_ABT1_EPP1008_0001 : EPP1008_78E8D3DD;
END_STRUCT
END_TYPE

// ---- DUTs/IO/Topology/R10_A3_EK1122_6A26DC25.TcDUT
{attribute 'GeneratedUsingTerminal: EK1122-0000-0018'}
{attribute addProperty BoxType "EK1122-0000-0018"}
{attribute addProperty Id "R10_AB00_EPP1322_0001R10_AB00_EPP1322_0001_481BC624168R10_AB1_EPP1008_0001EPP1008_78E8D3DD12R10_AB2_EPP1008_0001EPP1008_78E8D3DD12R10_AB3_EPP1008_0001EPP1008_78E8D3DD12R10_AB4_EPP1008_0001EPP1008_78E8D3DD12R10_AB5_EPP1008_0001EPP1008_78E8D3DD12R10_AB6_EPP1008_0001EPP1008_78E8D3DD12R10_AB02_EPP1332_0001EPP1332_1FC0878B2R10_AB7_EPP1008_0001EPP1008_78E8D3DD12R10_AB8_EPP1008_0001EPP1008_78E8D3DD12R10_AB11_EPP2308_0001EPP2308_F6D9A8D112R10_AB12_EPP2308_0001EPP2308_F6D9A8D112R10_AB13_EPP2308_0001EPP2308_F6D9A8D112"}
{attribute addProperty CRC "1780931621"}
{attribute addProperty Size "302"}
{attribute addProperty Name "R10_A3 (EK1122)"}
TYPE R10_A3_EK1122_6A26DC25 EXTENDS EK1122_1FC0878B :
STRUCT
    {attribute addProperty Name "R10-AB00 (EPP1322-0001)"}
    {attribute addProperty PreviousPort "R10_A3 (EK1122) : D"}
    {attribute addProperty SyncUnit "default"}
    R10_AB00_EPP1322_0001 : R10_AB00_EPP1322_0001_481BC624;
    {attribute addProperty Name "R10-AB1 (EPP1008-0001)"}
    {attribute addProperty PreviousPort "R10-AB00 (EPP1322-0001) : C"}
    {attribute addProperty SyncUnit "R10"}
    R10_AB1_EPP1008_0001 : EPP1008_78E8D3DD;
    {attribute addProperty Name "R10-AB2 (EPP1008-0001)"}
    {attribute addProperty PreviousPort "R10-AB1 (EPP1008-0001) : B"}
    {attribute addProperty SyncUnit "R10"}
    R10_AB2_EPP1008_0001 : EPP1008_78E8D3DD;
    {attribute addProperty Name "R10-AB3 (EPP1008-0001)"}
    {attribute addProperty PreviousPort "R10-AB2 (EPP1008-0001) : B"}
    {attribute addProperty SyncUnit "R10"}
    R10_AB3_EPP1008_0001 : EPP1008_78E8D3DD;
    {attribute addProperty Name "R10-AB4 (EPP1008-0001)"}
    {attribute addProperty PreviousPort "R10-AB3 (EPP1008-0001) : B"}
    {attribute addProperty SyncUnit "R10"}
    R10_AB4_EPP1008_0001 : EPP1008_78E8D3DD;
    {attribute addProperty Name "R10-AB5 (EPP1008-0001)"}
    {attribute addProperty PreviousPort "R10-AB4 (EPP1008-0001) : B"}
    {attribute addProperty SyncUnit "R10"}
    R10_AB5_EPP1008_0001 : EPP1008_78E8D3DD;
    {attribute addProperty Name "R10-AB6 (EPP1008-0001)"}
    {attribute addProperty PreviousPort "R10-AB5 (EPP1008-0001) : B"}
    {attribute addProperty SyncUnit "R10"}
    R10_AB6_EPP1008_0001 : EPP1008_78E8D3DD;
    {attribute addProperty Name "R10-AB02 (EPP1332-0001)"}
    {attribute addProperty PreviousPort "R10-AB6 (EPP1008-0001) : B"}
    {attribute addProperty SyncUnit "default"}
    R10_AB02_EPP1332_0001 : EPP1332_1FC0878B;
    {attribute addProperty Name "R10-AB7 (EPP1008-0001)"}
    {attribute addProperty PreviousPort "R10-AB02 (EPP1332-0001) : C"}
    {attribute addProperty SyncUnit "R10"}
    R10_AB7_EPP1008_0001 : EPP1008_78E8D3DD;
    {attribute addProperty Name "R10-AB8 (EPP1008-0001)"}
    {attribute addProperty PreviousPort "R10-AB7 (EPP1008-0001) : B"}
    {attribute addProperty SyncUnit "R10"}
    R10_AB8_EPP1008_0001 : EPP1008_78E8D3DD;
    {attribute addProperty Name "R10-AB11 (EPP2308-0001)"}
    {attribute addProperty PreviousPort "R10-AB8 (EPP1008-0001) : B"}
    {attribute addProperty SyncUnit "R10"}
    R10_AB11_EPP2308_0001 : EPP2308_F6D9A8D1;
    {attribute addProperty Name "R10-AB12 (EPP2308-0001)"}
    {attribute addProperty PreviousPort "R10-AB11 (EPP2308-0001) : B"}
    {attribute addProperty SyncUnit "R10"}
    R10_AB12_EPP2308_0001 : EPP2308_F6D9A8D1;
    {attribute addProperty Name "R10-AB13 (EPP2308-0001)"}
    {attribute addProperty PreviousPort "R10-AB12 (EPP2308-0001) : B"}
    {attribute addProperty SyncUnit "R10"}
    R10_AB13_EPP2308_0001 : EPP2308_F6D9A8D1;
END_STRUCT
END_TYPE

// ---- DUTs/IO/Topology/R10_EK1100_C5CE1D87.TcDUT
{attribute 'GeneratedUsingTerminal: EK1100-0000-0018'}
{attribute addProperty BoxType "EK1100-0000-0018"}
{attribute addProperty Id "R10_A2_EK1122R10_A2_EK1122_75D61001165R10_A3_EK1122R10_A3_EK1122_6A26DC25302R10_A4_EL6631EL6631_A0EC075C2R10_A4_EL7041_1000EL7041_86DE63E743R10_A5_EL1809EL1809_32157CFD20R10_A6_EL2809EL2809_2B6483BD19R10_A7_EL2809EL2809_2B6483BD19R10_A8_EL3024EL3024_C6E76B5A40R10_A9_EL1809EL1809_32157CFD20R10_A10_EL2809EL2809_2B6483BD19R10_EndTerminal_EL9011EL9011_D65D3D320"}
{attribute addProperty CRC "3318619527"}
{attribute addProperty Size "649"}
{attribute addProperty Name "R10 (EK1100)"}
TYPE R10_EK1100_C5CE1D87 EXTENDS EK1100_1FC0878B :
STRUCT
    {attribute addProperty Name "R10_A2 (EK1122)"}
    {attribute addProperty PreviousPort "R10 (EK1100) : B"}
    {attribute addProperty SyncUnit "default"}
    R10_A2_EK1122 : R10_A2_EK1122_75D61001;
    {attribute addProperty Name "R10_A3 (EK1122)"}
    {attribute addProperty PreviousPort "R10_A2 (EK1122) : C"}
    {attribute addProperty SyncUnit "default"}
    R10_A3_EK1122 : R10_A3_EK1122_6A26DC25;
    {attribute addProperty Name "R10_A4 (EL6631)"}
    {attribute addProperty PreviousPort "R10_A3 (EK1122) : C"}
    {attribute addProperty SyncUnit "R10"}
    R10_A4_EL6631 : EL6631_A0EC075C;
    {attribute addProperty Name "R10_A4 (EL7041-1000)"}
    {attribute addProperty PreviousPort "R10_A4 (EL6631) : B"}
    {attribute addProperty SyncUnit "R10"}
    R10_A4_EL7041_1000 : EL7041_86DE63E7;
    {attribute addProperty Name "R10_A5 (EL1809)"}
    {attribute addProperty PreviousPort "R10_A4 (EL7041-1000) : B"}
    {attribute addProperty SyncUnit "R10"}
    R10_A5_EL1809 : EL1809_32157CFD;
    {attribute addProperty Name "R10_A6 (EL2809)"}
    {attribute addProperty PreviousPort "R10_A5 (EL1809) : B"}
    {attribute addProperty SyncUnit "R10"}
    R10_A6_EL2809 : EL2809_2B6483BD;
    {attribute addProperty Name "R10_A7 (EL2809)"}
    {attribute addProperty PreviousPort "R10_A6 (EL2809) : B"}
    {attribute addProperty SyncUnit "R10"}
    R10_A7_EL2809 : EL2809_2B6483BD;
    {attribute addProperty Name "R10_A8 (EL3024)"}
    {attribute addProperty PreviousPort "R10_A7 (EL2809) : B"}
    {attribute addProperty SyncUnit "R10"}
    R10_A8_EL3024 : EL3024_C6E76B5A;
    {attribute addProperty Name "R10_A9 (EL1809)"}
    {attribute addProperty PreviousPort "R10_A8 (EL3024) : B"}
    {attribute addProperty SyncUnit "R10"}
    R10_A9_EL1809 : EL1809_32157CFD;
    {attribute addProperty Name "R10_A10 (EL2809)"}
    {attribute addProperty PreviousPort "R10_A9 (EL1809) : B"}
    {attribute addProperty SyncUnit "R10"}
    R10_A10_EL2809 : EL2809_2B6483BD;
    {attribute addProperty Name "R10_EndTerminal (EL9011)"}
    {attribute addProperty PreviousPort "R10_A10 (EL2809) : B"}
    {attribute addProperty SyncUnit "default"}
    R10_EndTerminal_EL9011 : EL9011_D65D3D32;
END_STRUCT
END_TYPE

// ---- DUTs/IO/Topology/Device_4_EtherCAT_07442C6B.TcDUT
{attribute 'GeneratedUsingTerminal: IODEVICETYPE_ETHERCATPROT'}
{attribute addProperty BoxType "IODEVICETYPE_ETHERCATPROT"}
{attribute addProperty Id "R1_EK1100R1_EK1100_4AD22B7B1143R2_EK1100R2_EK1100_10D8A594458R3_EK1100R3_EK1100_C7887D6C263R4_EK1100R4_EK1100_46A1248C369R4A_EK1100R4A_EK1100_48316913274R5_EK1100R5_EK1100_0007A337146R6_EK1100R6_EK1100_8C41F5F2336R7_EK1100R7_EK1100_F50DDAC8306R8_EK1100R8_EK1100_9C7B3B675648R9_EK1100R9_EK1100_484053C0136R10_EK1100R10_EK1100_C5CE1D87649SyncUnitsSyncUnits_5BE71B8B288InputsInputs_A65FACA410OutputsOutputs_23C0ED1D6InfoDataInfoData_84133AC922"}
{attribute addProperty CRC "121908331"}
{attribute addProperty Size "10054"}
{attribute addProperty Name "Device 4 (EtherCAT)"}
TYPE Device_4_EtherCAT_07442C6B EXTENDS TcoIo.EtcMasterBase_62654B43 :
STRUCT
    {attribute addProperty Name "R1 (EK1100)"}
    {attribute addProperty PreviousPort "Device 4 (EtherCAT) : Master"}
    {attribute addProperty SyncUnit "default"}
    R1_EK1100 : R1_EK1100_4AD22B7B;
    {attribute addProperty Name "R2 (EK1100)"}
    {attribute addProperty PreviousPort "R1 (EK1100) : C"}
    {attribute addProperty SyncUnit "default"}
    R2_EK1100 : R2_EK1100_10D8A594;
    {attribute addProperty Name "R3 (EK1100)"}
    {attribute addProperty PreviousPort "R2 (EK1100) : C"}
    {attribute addProperty SyncUnit "default"}
    R3_EK1100 : R3_EK1100_C7887D6C;
    {attribute addProperty Name "R4 (EK1100)"}
    {attribute addProperty PreviousPort "R3 (EK1100) : C"}
    {attribute addProperty SyncUnit "default"}
    R4_EK1100 : R4_EK1100_46A1248C;
    {attribute addProperty Name "R4A (EK1100)"}
    {attribute addProperty PreviousPort "R4 (EK1100) : C"}
    {attribute addProperty SyncUnit "default"}
    R4A_EK1100 : R4A_EK1100_48316913;
    {attribute addProperty Name "R5 (EK1100)"}
    {attribute addProperty PreviousPort "R4A (EK1100) : C"}
    {attribute addProperty SyncUnit "default"}
    R5_EK1100 : R5_EK1100_0007A337;
    {attribute addProperty Name "R6 (EK1100)"}
    {attribute addProperty PreviousPort "R5 (EK1100) : C"}
    {attribute addProperty SyncUnit "default"}
    R6_EK1100 : R6_EK1100_8C41F5F2;
    {attribute addProperty Name "R7 (EK1100)"}
    {attribute addProperty PreviousPort "R6 (EK1100) : C"}
    {attribute addProperty SyncUnit "default"}
    R7_EK1100 : R7_EK1100_F50DDAC8;
    {attribute addProperty Name "R8 (EK1100)"}
    {attribute addProperty PreviousPort "R7 (EK1100) : C"}
    {attribute addProperty SyncUnit "default"}
    R8_EK1100 : R8_EK1100_9C7B3B67;
    {attribute addProperty Name "R9 (EK1100)"}
    {attribute addProperty PreviousPort "R8 (EK1100) : C"}
    {attribute addProperty SyncUnit "default"}
    R9_EK1100 : R9_EK1100_484053C0;
    {attribute addProperty Name "R10 (EK1100)"}
    {attribute addProperty PreviousPort "R9 (EK1100) : C"}
    {attribute addProperty SyncUnit "default"}
    R10_EK1100 : R10_EK1100_C5CE1D87;
    {attribute addProperty Name "SyncUnits"}
    SyncUnits : SyncUnits_5BE71B8B;
    {attribute addProperty Name "Inputs"}
    Inputs : TcoIo.Inputs_A65FACA4;
    {attribute addProperty Name "Outputs"}
    Outputs : TcoIo.Outputs_23C0ED1D;
    {attribute addProperty Name "InfoData"}
    InfoData : TcoIo.InfoData_84133AC9;
END_STRUCT
END_TYPE

